# B&R Automation Studio project PLC code - cp (part 12)

#### BlockAlarms.st
```iecst
ACTION BlockAlarms:

	// Report alrms if is enabled. It comes from 4.3.6
	IF NOT Block.Status.xEnabledMovements THEN
		// Emergency stop alarm report to SW with block disabled
		SafetyEmergencyStopAlarms;
		RETURN;
	END_IF

	SafetyAlarms;

	ModulesElementsAlarms;

	VerticalMotorAlarms;

	CleanAlarms;

	//########################## ALARMS SUMMARY ########################################
	AlarmsSummary;

END_ACTION

ACTION SafetyAlarms:

	SafetyEmergencyStopAlarms;

	// Alarm: Curtain Alarm

	//[RGP]CRETALEGO-1297: Front curtain alarm always activated when conditions are TRUE. Not autoreset as previously.
	//Will be reset BY "ResetAlarms.st" when "Reset" button is pressed and conditions are no longer TRUE.
	//These lines have been moved up, before calling "T_SafetyError()", this way we can set the alarm before switching to ZERO state
	IF NOT Block.In.Safety.xCurtainEnable01 OR NOT Block.In.Safety.xCurtainEnable02 THEN
		Block.Al.xAlrFrontCurtain:= TRUE;
	END_IF

	//Alarm: Front and rear general alarm (from preventa)
	IF (NOT Block.In.Safety.xRearSafetyOK) THEN
		Block.Al.xAlrRearSafety:= TRUE;
	END_IF
	IF (NOT Block.In.Safety.xFrontSafetyOK) THEN
		Block.Al.xAlrFrontSafety:= TRUE;
	END_IF

	//Bars Out sensor Cube
	IF NOT Block.In.xBarsIn AND Block.Status.Motor.xBarsHomed THEN
		Block.Al.xAlrBarsOut := TRUE;
	END_IF

	//Any Upper Safety. Variable to better readin and reduce number of lines
	xAnyUpperSafety := Block.Al.xAlrFrontCurtain OR Block.Al.xAlrRearSafety OR Block.Al.xAlrFrontSafety OR Block.Al.xAlrBarsOut;

	// Safety feedback is down? Has it been validate by reset panel?
	//Used a TOF to avoid false signal when entering in AutoMode ALX check in P4 this functionallity
	T_SafetyError.IN:=	(NOT Block.commands.Mode.xZero) AND
						(xAnyUpperSafety OR Block.Al.xAlrEmergencyStop OR NOT Block.In.Safety.xSafetyOK) AND
						(NOT Block.commands.AutoMode.xBypass);

	T_SafetyError.PT:=t#150ms;
	T_SafetyError();

	IF T_SafetyError.Q THEN
		Block.Al.xAlrSafetySystemInBlock:= TRUE;
	END_IF

END_ACTION

ACTION SafetyEmergencyStopAlarms:

	CASE Block.parameters.Hw.SafetySignals OF
		SAFETY_ESTOP_CONNECTED:

			// Alarm: Emergency Stop Button
			IF NOT Block.In.Safety.xFrontEStopOK THEN
				Block.Al.xAlrFrontEmergencyStop := TRUE;
			END_IF

			IF NOT Block.In.Safety.xRearEStopOK THEN
				Block.Al.xAlrRearEmergencyStop:= TRUE;
			END_IF

			Block.Al.xAlrEmergencyStop := Block.Al.xAlrFrontEmergencyStop OR Block.Al.xAlrRearEmergencyStop;

		SAFETY_ESTOP_CALCULATED:

			//If we do not have Safety OK buy the upper safety is OK, it is considered and EStop button is pressed
			IF NOT Block.In.Safety.xSafetyOK AND Block.In.Safety.xFrontSafetyOK AND Block.In.Safety.xRearSafetyOK THEN
				Block.Al.xAlrLogicEmergencyStop:= TRUE;
			END_IF

			Block.Al.xAlrEmergencyStop := Block.Al.xAlrLogicEmergencyStop;

	END_CASE

END_ACTION

ACTION VerticalMotorAlarms:

	// Alarm: Not homed Vertical motor.
	Block.Al.xAlrBarMtrNoRef:= NOT Block.Status.Motor.xBarsHomed;

	// Alarm: Drive protection
	IF NOT Block.In.xDriveProtectionOK THEN
		Block.Al.xAlrDriveProtection:= TRUE;
	END_IF

	// Alarm: Temp Vertical Motor
	IF AxisBK.Status.ActTempMot > (AxisBK.Status.MaxTempMotor - 5.0) THEN
		Block.Al.xBarMotorTemp := TRUE;
	ELSIF AxisBK.Status.ActTempMot < (AxisBK.Status.MaxTempMotor - 7.0) THEN
		Block.Al.xBarMotorTemp := FALSE;
	END_IF

	// Alarm: Temp Vertical Driver
	IF AxisBK.Status.ActTempDrv > (AxisBK.Status.MaxTempDrv - 5.0) THEN
		Block.Al.xBarDriverTemp := TRUE;
	ELSIF AxisBK.Status.ActTempDrv < (AxisBK.Status.MaxTempDrv - 7.0) THEN
		Block.Al.xBarDriverTemp := FALSE;
	END_IF

	//Alarm: Comms error in Vertical motor
	// Pass codes to ennum type 32189
	IF (AxisBK.Status.ErrorID=29265) OR (AxisBK.Status.ErrorID=32189) THEN
		Block.Al.xAlrComBarMtr:= TRUE;
	END_IF

	// Alarm: Any drive Alarm
	TON_DelayAnyVerticalDriveAlarm.IN:= AxisBK.Status.ErrorID<>0 AND
										NOT Block.AlSummary.xAlrSafetySystemGeneral AND
										NOT Block.commands.Mode.xZero AND
										NOT xAnyUpperSafety;
	TON_DelayAnyVerticalDriveAlarm.PT:=t#200ms;
	TON_DelayAnyVerticalDriveAlarm();
	IF TON_DelayAnyVerticalDriveAlarm.Q THEN
		ReasonErrorID := AxisBK.Status.ErrorID;
		Block.Al.xAnyVerticalDriveAlarm:= TRUE;
	END_IF

	// Alarm: Power Error
	//[RGP] Power mains: At least one phase of the power line failed
	IF AxisBK.Status.ErrorID=7215 THEN
		Block.Al.xAlBarMotorPowerOff:= TRUE;
	END_IF

	// Warning: Decrease clean offset.
	TOF_CleanOffsetChng.IN := rOffseCleanMtr <> rOffseCleanMtr_Copy;
	TOF_CleanOffsetChng.PT := t#10s;
	TOF_CleanOffsetChng();
	Block.Al.xAlrDecreaseCleanOffset:= TOF_CleanOffsetChng.Q;

	//Warning: Check Homing Sensor Broken
	IF Block.Al.xAnyVerticalDriveAlarm AND (Block.Status.PositionState = BLOCKP_HOMING_BAR) THEN
		Block.Al.xAlrCheckHomingSensor:=TRUE;
	END_IF

	// Warning: Vertical motor maxium lifting alarm
	IF rMotorCurrentPos >= Block.parameters.Motor.rSafePosition THEN
		Block.Al.xAlrBlockReachedMaxPosition := TRUE;
	END_IF

	// Warning: Reference incoherence or broken reference sensor wire
	T_DelayAlarmRef.IN:=Block.In.xReferenceDI <> AxisBK.Status.DigitalInputs.RefSwitch;
	T_DelayAlarmRef.PT:=T#500ms;
	T_DelayAlarmRef();

	IF T_DelayAlarmRef.Q THEN
		Block.Al.xAlrReferenceIncoherence := TRUE;
	END_IF

	//Critical: Controller Not Ready
	ton_ControllerReady.IN := (NOT AxisBK.Status.ControllerReady OR AxisBK.Status.ErrorID=6029 OR AxisBK.Status.ErrorID=29216) AND NOT Block.commands.Mode.xZero;	//ErrorID 6029 its for motors with breaker and ControllerReady its general
	ton_ControllerReady.PT := t#300ms;																																//ErrorID 29216 to detect just power wires disconected
	ton_ControllerReady();
	IF ton_ControllerReady.Q THEN
		Block.Al.xAlrControllerNotReady := TRUE;
	END_IF

	//Warning Over Torque
	TON_OvertorqueWarning.IN := ABS(AxisBK.Status.ActTorque) > (Block.Status.Motor.rOperationTorque); //AxisBK.Status.RatedTorque;
	TON_OvertorqueWarning.PT := T#10s; //T#2s;
	TON_OvertorqueWarning();

	IF TON_OvertorqueWarning.Q THEN
		Block.Al.xWrnOverTorq := TRUE;
	END_IF

	// Alarm: Over Torque
	tonOvertorqueAlarm.IN := ABS(AxisBK.Status.ActTorque) > (1.6*Block.Status.Motor.rOperationTorque); //(AxisBK.Status.RatedTorque);
	tonOvertorqueAlarm.PT := T#500ms;	//T#5s;
	tonOvertorqueAlarm();
	IF tonOvertorqueAlarm.Q THEN
		Block.Al.xAlrOverTorque := TRUE;
	END_IF

	//Alarms related to collision between bars and tray
	CASE Block.Status.PositionState OF
		BLOCKP_UNDEFINED,
		BLOCKP_IN_CAP,
		BLOCKP_IN_CLEAN,
		BLOCKP_HOMING_ICLA:
			// Do nothing

		BLOCKP_IN_PRINT:
			//Raise warning and alarm if the tray sensor is disconected while in risk position (below dripping position)
			tonDelayTraySensorError.IN := NOT Block.In.xTrayOut;
			tonDelayTraySensorError.PT := T#750ms;
			tonDelayTraySensorError();

			//Raise asking the machine to emptyBelt
			IF tonDelayTraySensorError.Q AND Block.parameters.xMediaBelow THEN
				Block.Status.xAlarmToEmptyBelt := TRUE;
			//Raise and stop alarm once the belt is empty
			ELSIF tonDelayTraySensorError.Q AND NOT Block.parameters.xMediaBelow THEN
				Block.Al.xAlrTraySensor:=TRUE;
				Block.Status.xAlarmToEmptyBelt := FALSE;
			END_IF

		BLOCKP_GOING_TO_CAP,
		BLOCKP_GOING_TO_PRINT,
		BLOCKP_GOING_TO_CLEAN,
		BLOCKP_CLEANING,
		BLOCKP_HOMING_BAR:
			//Risk. Moving!
			xDangerCollision := NOT Block.In.xTrayOut OR NOT Block.In.xIclaSensor;
			IF NOT Block.In.xTrayOut AND 	(((rMotorCurrentPos<Block.parameters.Motor.rDripBarsPosition) AND NOT Block.parameters.xCappingProcess) OR
												(rMotorCurrentPos<Block.parameters.Motor.rCappingPosition)) OR

				NOT Block.In.xIclaSensor AND (((rMotorCurrentPos<Block.parameters.Motor.rSafePositionCleanCarrier) AND NOT Block.parameters.xCappingProcess) OR
												(rMotorCurrentPos<Block.parameters.Motor.rCappingPosition))	THEN

					Block.Al.xNoActionDangerCollision:=TRUE;
			END_IF
	END_CASE

	//Saving state where alarm was raised
	IF EDGEPOS(Block.Al.xNoActionDangerCollision) THEN
		iReasonDanger.0:=NOT Block.In.xTrayOut;
		iReasonDanger.1:=NOT Block.In.xIclaSensor;

		nStateDanger := nState;
		PositionStateDanger:=Block.Status.PositionState;
	END_IF

	//If the sensor is conected again. Remove the memory
	IF Block.In.xTrayOut THEN
		Block.Status.xAlarmToEmptyBelt := FALSE;
	END_IF

END_ACTION

ACTION ModulesElementsAlarms:

	// Alarm: Differential NOK
	IF NOT Block.In.xDifferentialOK THEN
		Block.Al.xAlrDif:= TRUE;
	END_IF

	// Alarm: TempPowerSupply
	IF Block.parameters.Hw.iNumHeaterPSU>0 THEN
		Block.Al.xAlrTempPowerSupply:= FALSE;
		FOR iIndexPsu:=1 TO Block.parameters.Hw.iNumHeaterPSU DO
			IF NOT Block.In.xHeaterDcOkPsu[iIndexPsu] OR NOT Block.In.xHeaterAcOkPsu[iIndexPsu] THEN
				Block.Al.xAlrTempPowerSupply:= TRUE;
			END_IF
		END_FOR

		IF NOT Block.In.xHeaterDcOkBusBar1 OR NOT Block.In.xHeaterDcOkBusBar2 THEN
			Block.Al.xAlrTempPowerSupply:= TRUE;
		END_IF
	END_IF

	// Logging the exact signal that raises the Heaters Power supply alarm
	IF EDGENEG(Block.In.xHeaterDcOkBusBar1) THEN LogErrorxHeaterDcOkBusBar1; END_IF
	IF EDGENEG(Block.In.xHeaterDcOkBusBar2) THEN LogErrorxHeaterDcOkBusBar2; END_IF
	IF EDGENEG(Block.In.xHeaterDcOkPsu[1]) THEN LogErrorxHeaterDcOkPsu1; END_IF
	IF EDGENEG(Block.In.xHeaterDcOkPsu[2]) THEN LogErrorxHeaterDcOkPsu2; END_IF
	IF EDGENEG(Block.In.xHeaterDcOkPsu[3]) THEN LogErrorxHeaterDcOkPsu3; END_IF
	IF EDGENEG(Block.In.xHeaterAcOkPsu[1]) THEN LogErrorxHeaterAcOkPsu1; END_IF
	IF EDGENEG(Block.In.xHeaterAcOkPsu[2]) THEN LogErrorxHeaterAcOkPsu2; END_IF
	IF EDGENEG(Block.In.xHeaterAcOkPsu[3]) THEN LogErrorxHeaterAcOkPsu3; END_IF

	// Alarm: PrintHead PowerSupply
	IF Block.parameters.Hw.iNumPrintheadsPSU>0 THEN
		Block.Al.xAlrPHPowerSupply:= FALSE;
		FOR iIndexPsu:=1 TO Block.parameters.Hw.iNumPrintheadsPSU DO
			IF NOT Block.In.xPrintHeadPSU[iIndexPsu] THEN
				Block.Al.xAlrPHPowerSupply:= TRUE;
			END_IF
		END_FOR
	END_IF

	// Alarm: Module Temp 01
	Block.Al.xModuleTemp01:= NOT Block.In.xModuleTemp01Ok;

	// Alarm: Module Temp 02
	Block.Al.xModuleTemp02:= NOT Block.In.xModuleTemp02Ok;

	// Alarm: Module Temp 03
	Block.Al.xModuleTemp03:= NOT Block.In.xModuleTemp03Ok AND Block.parameters.Inks.xTankHeatEnabled1;

	// Alarm: Module Temp 04
	Block.Al.xModuleTemp04:= NOT Block.In.xModuleTemp04Ok AND Block.parameters.Inks.xTankHeatEnabled2;

	(*SI UNIT ALARMS*)
	//Alarm venturi
	IF NOT Block.In.xAirVenturiOK AND Block.In.xSiUnitModuleOk THEN
		Block.Al.xAlAirVenturi:= TRUE;
	END_IF

	// Alarm: Coms error SI Unit
	IF NOT Block.In.xSiUnitModuleOk  THEN
		Block.Al.xAlrComSiUnit:= TRUE;
		Block.Al.xSiUnitPowerOff:=TRUE;
	END_IF

END_ACTION

ACTION CleanAlarms:

	// Warning: Alarms of no action allowed due to colision warning.
	Block.Al.xAlrNoTrayInServoNoHomed:=(NOT AxisBK.Status.HomeOK) AND Block.commands.Manual.xManTrayIn;

	// Warning: clean interrupt
	Block.Al.xAlCleanInterrupt:= xCleanInterrupt;

	// ICLA		ICLA		ICLA		ICLA		ICLA		ICLA		ICLA		ICLA
	// ICLA		ICLA		ICLA		ICLA		ICLA		ICLA		ICLA		ICLA

	//Alarm: Comms error in cleaning motor
	T_AlrComsCleanMotor.IN:= NOT IclaBK.Status.xModuleOK;
	T_AlrComsCleanMotor.PT:= T#2S;
	T_AlrComsCleanMotor();

	IF T_AlrComsCleanMotor.Q THEN
		Block.Al.xAlrComCleanMtr:= TRUE;
	END_IF

	//Alarm: Not homed cleaning motor.
	Block.Al.xAlrCleanMtrNoRef:= NOT Block.Status.Icla.xHomed;

	// From Icla error table 011Ah 282 4 Inputs of the STO safety function have different levels (>1s). Reset done executing ResetAlarms in Machine program
	// If the connector is removed while moving is error 281, error 282 is STO at different level
	IF (IclaBK.Status.Error.ErrorNumber = 281 OR IclaBK.Status.Error.ErrorNumber = 282) THEN
		Block.Al.xAlrEnabCleanMtrDiffLvL:= TRUE;
	END_IF

	// Alarm: Any clean motor alarm
	T_IclaError.IN :=	(IclaBK.Status.Error.ErrorNumber<>0 OR IclaBK.Status.iDriveStatus = ICLAST_SWITCH_ON_DISABLED OR IclaBK.Status.iDriveStatus = ICLAST_ERROR) AND
						Block.In.Safety.xSafetyOK AND
						NOT Block.AlSummary.xAlrSafetySystemGeneral AND //This variable must not be required so we already check "Block.In.Safety.xSafetyOK"
						NOT Block.commands.Mode.xZero AND
						NOT xAnyUpperSafety; //This variable must not be required so we already check "Block.In.Safety.xSafetyOK"
	T_IclaError.PT := t#250ms;
	T_IclaError();
	IF T_IclaError.Q THEN
		Block.Al.xAlrCleanMotor:= TRUE;
	END_IF

	Block.Al.xCleanMotorControllerNotReady := IclaBK.Status.iDriveStatus = ICLAST_SWITCH_ON_DISABLED AND Block.In.Safety.xSafetyOK AND NOT Block.commands.Mode.xZero;

	// Alarm: Clean Sensor
	T_AlCleanSensor.IN:= Block.Status.Icla.xHomed AND (NOT Block.In.xIclaSensor) AND (rIclaCurrentPos<=0) AND Block.In.xSiUnitModuleOk;
	T_AlCleanSensor.PT:= t#2500ms;
	T_AlCleanSensor();
	IF T_AlCleanSensor.Q THEN
		Block.Al.xAlrCleanSensor:= TRUE;
	END_IF

	// TRAY ALARMS		TRAY ALARMS		TRAY ALARMS		TRAY ALARMS		TRAY ALARMS		TRAY ALARMS		TRAY ALARMS		TRAY ALARMS
	// TRAY ALARMS		TRAY ALARMS		TRAY ALARMS		TRAY ALARMS		TRAY ALARMS		TRAY ALARMS		TRAY ALARMS		TRAY ALARMS

	TNotPrinterZero.IN:=NOT (Block.commands.Mode.xZero);
	TNotPrinterZero.PT:=T#500ms;
	TNotPrinterZero();

	//This is to avoid alarms in Zero mode when manually moving the tray
	IF TNotPrinterZero.Q THEN
		TON_AlrTrayIn(IN := Block.Out.xTrayIn, PT:= Block.parameters.tiTimeWaitTrayInAlarm);
		TON_AlrTrayOut(IN := Block.Out.xTrayOut, PT:= Block.parameters.tiTimeWaitTrayOutAlarm);
	END_IF

	// Alr tray sensor IN
	IF TON_AlrTrayIn.Q AND (NOT Block.In.xTrayIn) THEN
		Block.Al.xAlrTraySensor:=TRUE;
	END_IF
	// Alr tray sensor OUT
	IF TON_AlrTrayOut.Q AND (NOT Block.In.xTrayOut) THEN
		Block.Al.xAlrTraySensor:=TRUE;
	END_IF

	//Alarm clean motor ERROR POSITION// issue 1269
	T_DelayIncoherCleanMtr.IN :=	((nState=233 AND NOT Block.In.xIclaSensor) OR
									(rIclaCurrentPos>LIMITPOSINCOHERCLEANMOTOR AND Block.In.xIclaSensor));
	T_DelayIncoherCleanMtr.PT:= T#500MS;
	T_DelayIncoherCleanMtr();

	IF T_DelayIncoherCleanMtr.Q THEN
		Block.Al.xAlrIncoherPositCleanMtr:= TRUE;
	END_IF
	//Poner aquí la gestion de las alarmas y, si eso, sacar la habilitación fuera, ya que no es su sitio
	//Secuencia - Alarmas de tanque y bomba - Sirena - Hab/Deshab - parada a mitad de proceso - ....

	//If Machine are Water enable water alarms
	IF Block.Status.xIsWaterBlock THEN

		//Water tank empty alarm
		IF NOT Block.In.xWaterLevelSensor THEN
			Block.Al.xAlrEmptyWaterTank:=TRUE;
		END_IF

		//Water Presure and broken presure sensor alarms
		T_AlrNoPressureWhenWaterPumpIsOn.IN:=Block.Out.xCleaningWaterPump AND Block.In.xWaterPresureSensor;
		T_AlrNoPressureWhenWaterPumpIsOn.PT:=T#5S;
		T_AlrNoPressureWhenWaterPumpIsOn();
		IF T_AlrNoPressureWhenWaterPumpIsOn.Q THEN
			Block.Al.xAlrWaterPumpPresure:=TRUE;
		END_IF

		//Broquen wire or pressure switch not work alarm
		IF NOT Block.In.xWaterPresureSensor AND NOT Block.Out.xCleaningWaterPump AND NOT nState=264 THEN
			Block.Al.xAlrWtrPresSensBroken := TRUE;
		END_IF

		//Capping water Alarms:
		//Water flowmeter and WaterTankEmpty
		IF Block.parameters.xCappingProcess  THEN

			//Water tank empty alarm
			IF NOT Block.In.xCappingWaterLevelSensor THEN
				Block.Al.xAlrCappingWaterTankEmpty:=TRUE;
			END_IF

			//Water recirculation alarm
			TON_AlrCappingWaterNotRecirc.IN:=(Block.Out.xCappingWaterPump AND NOT Block.In.xCappingWaterFlowmeter);
			TON_AlrCappingWaterNotRecirc.PT:=T#3S;
			TON_AlrCappingWaterNotRecirc();

			IF TON_AlrCappingWaterNotRecirc.Q THEN
				//Block.Al.xAlrCappingWaterNotRecirc:=TRUE;
			END_IF
		END_IF

	END_IF

	xAlrToAvoidCleanWithWater := Block.Al.xAlrEmptyWaterTank OR Block.Al.xAlrWaterPumpPresure OR Block.Al.xAlrWtrPresSensBroken;

END_ACTION
```

#### BlockManager.st
```iecst
PROGRAM _INIT
	FOR iIndexHistory:=0  TO iHistoryLines DO
		StateGenHistory[iIndexHistory]:=BLOCK_STOPPED;
		StatePosHistory[iIndexHistory]:=BLOCKP_UNDEFINED;
	END_FOR
END_PROGRAM

(*
PROGRAM _INIT

	//Define a transmision data to do the first calculations and be receptive to next calculations
	MotorDriveUnit.TransmissionData:=Block.parameters.Motor.DriveUnit;

	//Acceleration and deceleration
	MotorDriveUnit.AccelerationDesired := 10;
	MotorDriveUnit.Calculation := CALC_ACC_PULSES;
	MotorDriveUnit();

	MotorDriveUnit.DecelerationDesired := 10;
	MotorDriveUnit.Calculation := CALC_DEC_PULSES;
	MotorDriveUnit();

END_PROGRAM
*)

PROGRAM _CYCLIC

	// Block Reference
	Block ACCESS ADR(gBlock[gIndexBlock]);
	AxisBK ACCESS ADR (gAxis[Block.parameters.iMotorAxisIndex]);
	IclaBK ACCESS ADR (gIcla[Block.parameters.iIclaAxisIndex]);

	//If the Block doesn't exist, remove alarms and exit. Extra condition to avoid a divided by 0 error at start
	IF NOT Block.parameters.Hw.xExistBlock OR Block.parameters.Inks.iMaxBlockPrintBars = 0 THEN
		ResetAlarms;
		ResetBlockCommands;
		gIndexBlock := gIndexBlock + 1;
		RETURN;
	END_IF

	Inputs;

	//Limit the value of parameters configured
	BlockParameters;

	IF Block.parSw.xEnableToMovements THEN
		Block.Status.xEnabledMovements:= TRUE;
	ELSIF NOT Block.parSw.xEnableToMovements AND (xInCap OR NOT Block.Status.Motor.xBarsHomed) THEN
		Block.Status.xEnabledMovements:= FALSE;
	END_IF

	IF Block.commands.xReset THEN
		ResetAlarms;
	END_IF

	BlockAlarms;
	AlarmSound;

	IF (NOT Block.Status.xEnabledMovements) THEN
		gIndexBlock := gIndexBlock + 1;
		RETURN;
	END_IF

	GetInkSystemsData;

	ControlState;

	BlockStatesCtrl;

	AssignDataToInksSystem;

	InputParamsMotors;

	//Managment of the valves unit of the block. Reset if needed
	ValvesUnit;

	//Copy of variables to check changes
	rOffseCleanMtr_Copy:=rOffseCleanMtr;

	ResetEdgeCommands;

	//Increased exec times number to be checked outside
	Block.Status.execTimes := Block.Status.execTimes + 1;

	// Index added
	gIndexBlock := gIndexBlock + 1;

END_PROGRAM
```

#### BlockStateGen.st
```iecst
ACTION BlockStateGen:

	// PRINT POSITION ORDER
	xOrderToPrint:=	(Block.commands.xToPrint AND Block.parSw.xEnableToPrint) OR
					(Block.commands.xToPrintLab AND Block.commands.AutoMode.xLaboratory);

	// CAP POSITION ORDER
	//When in capping position, bars are touching the tray and was required to be able to move out bars in auto mode when front doors is opened
	IF Block.Status.Position.xInCap AND Block.parameters.xCappingProcess THEN
		xFrontDoorStatusChanged := (Block.In.xFrontDoorClosed <> xFrontDoorStatus) OR
									(NOT Block.In.xFrontDoorClosed AND EDGEPOS(Block.commands.Mode.xAuto));
	END_IF

	xCapOrder:= Block.commands.xToCap OR
				(Block.commands.xToCapLab AND Block.commands.AutoMode.xLaboratory) OR
				EDGENEG(Block.parSw.xEnableToPrint) OR
				xFrontDoorStatusChanged;

	xFrontDoorStatus := Block.In.xFrontDoorClosed;

	// CLEANING CYCLE FROM SW COMMAND
	Block.Status.xIsWaterBlock := Block.parameters.Hw.xIsWater AND Block.commands.xEnableCleaningWithWater;
	IF Block.Status.xIsWaterBlock AND xAlrToAvoidCleanWithWater THEN
		Block.Status.xEnabledToClean := FALSE;
	ELSE
		Block.Status.xEnabledToClean := TRUE;
	END_IF

	rsCleaning.SET:= Block.Status.xEnabledToClean AND
					(Block.commands.xStartToCleanOrder AND Block.Status.PositionState <> BLOCKP_CLEANING);
	rsCleaning.RESET1:= NOT Block.Status.xEnabledToClean OR
						EDGEPOS(Block.Status.xCleaningDone) OR
						NOT (Block.commands.Mode.xAuto);
	rsCleaning();
	xStartToCleanOrder:=rsCleaning.Q1;

	//To reset manual commands when not in manual mode
	IF Block.Status.BlockState <> BLOCK_MANUAL THEN
		Block.commands.Manual := ResetManCommands;
	END_IF

	CASE Block.Status.BlockState OF

		BLOCK_STOPPED:
			AxisBK.Command.QuickStop:=FALSE;

		BLOCK_STOPPING:
			StopMovements;
			//Added to modify block position so for example when homing icla or bar and
			//going TO zero, block position remained in homing even motors were stopped and Block status were "BLOCK_STOPPING"
			IF (Block.Status.PositionState=BLOCKP_HOMING_ICLA OR Block.Status.PositionState=BLOCKP_HOMING_BAR) THEN
				Block.Status.PositionState := BLOCKP_UNDEFINED;
			END_IF

			IF AllDevicedStopped(ADR(Block), ADR(AxisBK), ADR(IclaBK)) THEN
				Block.Status.BlockState := BLOCK_STOPPED;
			END_IF

		BLOCK_MANUAL:
			ManualMovements;

			IF Block.commands.xIclaHomeOrder AND NOT Block.Status.Motor.xBarsHoming THEN
				IF Block.parameters.xPrinterKeyMaintenanceActivated THEN
					Block.commands.xIclaHomeOrder:=FALSE;
				ELSE
					Block.Status.PositionState := BLOCKP_HOMING_ICLA;
				END_IF

			// To do home in block is mandatory to have Icla at sensor and try out
			ELSIF Block.commands.xBarHomeOrder THEN

				IF Block.In.xTrayIn OR NOT Block.In.xIclaSensor OR Block.parameters.xPrinterKeyMaintenanceActivated THEN
					Block.commands.xBarHomeOrder:=FALSE;
				ELSIF Block.In.xTrayOut AND Block.In.xIclaSensor AND NOT Block.Al.xAlrReferenceIncoherence THEN
					Block.Status.PositionState := BLOCKP_HOMING_BAR;
				ELSE
					Block.commands.xBarHomeOrder:=FALSE;
				END_IF

			ELSIF Block.commands.xToCleanPosition AND Block.Status.PositionState = BLOCKP_IN_CAP THEN
				Block.Status.PositionState := BLOCKP_GOING_TO_CLEAN;
				//Signal reseted outside the case to avoid a memory if the movement cannot be done

			ELSIF Block.commands.Manual.xToPrintPosition AND NOT Block.parameters.xMediaBelow AND Block.Status.PositionState = BLOCKP_IN_CAP THEN
				Block.Status.PositionState := BLOCKP_GOING_TO_PRINT;
				//Signal reseted outside the case to avoid a memory if the movement cannot be done

			END_IF

		BLOCK_AUTO:
			IF xStartToCleanOrder THEN

				//Enable cleaning in bar to end ReverseFlow
				IF Block.Status.PositionState <> BLOCKP_CLEANING THEN
					IF 	Block.Status.PositionState = BLOCKP_GOING_TO_PRINT OR Block.Status.PositionState = BLOCKP_IN_PRINT THEN
						BlockPositionPreviousCleaning := BLOCKP_GOING_TO_PRINT;
					ELSE
						BlockPositionPreviousCleaning := BLOCKP_GOING_TO_CAP;
					END_IF
					Block.Status.PositionState := BLOCKP_CLEANING;
				END_IF

				//If receiving a Going to Cap order while cleaning, store the information
				IF xCapOrder THEN
					BlockPositionPreviousCleaning := BLOCKP_GOING_TO_CAP;
				END_IF

			ELSIF (xCapOrder AND Block.Status.Motor.xBarsHomed AND (Block.In.xIclaSensor OR IclaBK.Status.iDriveStatus=ICLAST_ENABLE_OPERATION)) THEN
				//I move to STOP
				Block.Status.PositionState := BLOCKP_GOING_TO_CAP;

			ELSIF xOrderToPrint AND NOT xInPrint AND NOT Block.AlSummary.xAlarmCritical AND NOT Block.AlSummary.xAlarmStop THEN
				//Going TO PRINT
				Block.Status.PositionState := BLOCKP_GOING_TO_PRINT;

			END_IF

			IF 	EDGEPOS(Block.Status.xCleaningDone) THEN
				//Once he cleaning has finished, go to the previous position
				Block.Status.PositionState := BlockPositionPreviousCleaning;
			END_IF

	END_CASE

	//Copying block's outputs to status
	Block.Status.ManualCommands := Block.Out;

	//Saving state history
	IF Block.Status.BlockState<>StateGenHistory[0] THEN
		ShiftArrayForward(ADR(StateGenHistory), SIZEOF(StateGenHistory), SIZEOF(StateGenHistory[0]), 1, iHistoryLines);
		StateGenHistory[0]:=Block.Status.BlockState;
	END_IF

END_ACTION
```

#### EventLog.st
```iecst
ACTION LogCriticalAlarm:

//	iReasonCritical.0 := (Block.Al.xAlrSafetySystemInBlock AND Block.Status.xEnabledMovements);
//	iReasonCritical.1 := Block.Al.xAlrDif;
//	iReasonCritical.2 := Block.Al.xAlrDriveProtection;

	stEventLogCritical.Source := ELOG_TYPE_BLOCK;
	stEventLogCritical.Severity:= ELOG_SEVERITY_ERROR;
	stEventLogCritical.Facility:= gIndexBlock;
	stEventLogCritical.ErrorCode:=0;

	stEventLogCritical.Text := 'Block.LogCriticalAlarm';

	IF 		iReasonCritical.0 THEN stEventLogCritical.Text := 'Block. xAlrSafetySystemInBlock';
	ELSIF 	iReasonCritical.1 THEN stEventLogCritical.Text := 'Block. xAlrDif';
	ELSIF 	iReasonCritical.2 THEN stEventLogCritical.Text := 'Block. xAlrDriveProtection';
	END_IF

	gEventLogLoader(EventData := ADR(stEventLogCritical));

END_ACTION

ACTION LogStopAlarm:

	stEventLogStop.Source := ELOG_TYPE_BLOCK;
	stEventLogStop.Severity:= ELOG_SEVERITY_ERROR;
	stEventLogStop.Facility:= gIndexBlock;
	stEventLogStop.ErrorCode:=0;

	stEventLogStop.Text := 'Block.LogStopAlarm';

	IF 		iReasonStop.0 THEN stEventLogStop.Text := 'Block. xAlrCleanMtrNoRef';
	ELSIF 	iReasonStop.1 THEN stEventLogStop.Text := 'Block. xAlAirVenturi';
	ELSIF 	iReasonStop.2 THEN stEventLogStop.Text := 'Block. xAnyDriveAlarm';
	ELSIF 	iReasonStop.3 THEN stEventLogStop.Text := 'Block. xAlrBarMtrNoRef';
	ELSIF 	iReasonStop.4 THEN stEventLogStop.Text := 'Block. xSiUnitPowerOff';
	ELSIF 	iReasonStop.5 THEN stEventLogStop.Text := 'Block. xAlrComSiUnit';
	ELSIF 	iReasonStop.6 THEN stEventLogStop.Text := 'Block. xAlrComBarMtr';
	ELSIF 	iReasonStop.7 THEN stEventLogStop.Text := 'Block. xAlrCleanMotor';
	ELSIF 	iReasonStop.8 THEN stEventLogStop.Text := 'Block. xAlrComCleanMtr';
	ELSIF 	iReasonStop.9 THEN stEventLogStop.Text := 'Block. xAlrEnabCleanMtrDiffLvL';
	ELSIF 	iReasonStop.10 THEN stEventLogStop.Text := 'Block. xAlrIncoherPositCleanMtr';
	ELSIF 	iReasonStop.11 THEN stEventLogStop.Text := 'Block. xAlCleanInterrupt';
	ELSIF 	iReasonStop.12 THEN stEventLogStop.Text := 'Block. xAlrTrayCleanSensor';
	ELSIF 	iReasonStop.13 THEN stEventLogStop.Text := 'Block. xNoActionDangerCollision';
	ELSIF 	iReasonStop.14 THEN stEventLogStop.Text := 'Block. xAlrControllerNotReady';
	ELSIF 	iReasonStop.15 THEN stEventLogStop.Text := 'Block. xAlrOverTorque';
	END_IF

	//Adding nState data to log
	strAuxEventDesc := '. nSt= ';
	brsstrcat(ADR(stEventLogStop.Text), ADR(strAuxEventDesc));
	brsitoa(nState, ADR(strAuxEventDesc));
	brsstrcat(ADR(stEventLogStop.Text), ADR(strAuxEventDesc));
	strAuxEventDesc := '. nDg= ';
	brsstrcat(ADR(stEventLogStop.Text), ADR(strAuxEventDesc));
	brsitoa(nStateDanger, ADR(strAuxEventDesc));
	brsstrcat(ADR(stEventLogStop.Text), ADR(strAuxEventDesc));

	gEventLogLoader(EventData := ADR(stEventLogStop));

END_ACTION

ACTION LogToCapOrder:

	stEventLogToCap.Source := ELOG_TYPE_BLOCK;
	stEventLogToCap.Severity:= ELOG_SEVERITY_INFO;
	stEventLogToCap.Facility:= gIndexBlock;
	stEventLogToCap.ErrorCode:=0;

	stEventLogToCap.Text := 'Order to Cap BK: ';
	brsitoa(gIndexBlock, ADR(strAuxEventDesc));
	brsstrcat(ADR(stEventLogToCap.Text), ADR(strAuxEventDesc));

	gEventLogLoader(EventData := ADR(stEventLogToCap));

END_ACTION

ACTION LogToPrintOrder:

	stEventLogToPrint.Source := ELOG_TYPE_BLOCK;
	stEventLogToPrint.Severity:= ELOG_SEVERITY_INFO;
	stEventLogToPrint.Facility:= gIndexBlock;
	stEventLogToPrint.ErrorCode:=0;

	stEventLogToPrint.Text := 'Order to Print BK: ';
	brsitoa(gIndexBlock, ADR(strAuxEventDesc));
	brsstrcat(ADR(stEventLogToPrint.Text), ADR(strAuxEventDesc));

	gEventLogLoader(EventData := ADR(stEventLogToPrint));

END_ACTION

ACTION LogToCleanOrder:

	stEventLogToClean.Source := ELOG_TYPE_BLOCK;
	stEventLogToClean.Severity:= ELOG_SEVERITY_INFO;
	stEventLogToClean.Facility:= gIndexBlock;
	stEventLogToClean.ErrorCode:=0;

	stEventLogToClean.Text := 'Order to Clean BK: ';
	brsitoa(gIndexBlock, ADR(strAuxEventDesc));
	brsstrcat(ADR(stEventLogToClean.Text), ADR(strAuxEventDesc));

	gEventLogLoader(EventData := ADR(stEventLogToClean));

END_ACTION

ACTION LogVertMovementOrder:

	VerMotorEventLog.Source := ELOG_TYPE_BLOCK;
	VerMotorEventLog.Severity:= ELOG_SEVERITY_INFO;
	VerMotorEventLog.Facility:= gIndexBlock;
	VerMotorEventLog.ErrorCode:=0;

	VerMotorEventLog.Text := 'BK:';
	brsitoa(gIndexBlock, ADR(strAuxEventDesc));
	brsstrcat(ADR(VerMotorEventLog.Text), ADR(strAuxEventDesc));

	brsstrcat(ADR(VerMotorEventLog.Text), ADR(' from '));
	brsftoa(MotorDriveUnit.PositionDevice, ADR(strAuxEventDesc));
	brsstrcat(ADR(VerMotorEventLog.Text), ADR(strAuxEventDesc));

	brsstrcat(ADR(VerMotorEventLog.Text), ADR('mm to '));
	brsftoa(MotorDriveUnit.PositionDesired, ADR(strAuxEventDesc));
	brsstrcat(ADR(VerMotorEventLog.Text), ADR(strAuxEventDesc));

	brsstrcat(ADR(VerMotorEventLog.Text), ADR('mm at '));
	brsftoa(MotorDriveUnit.SpeedDesired, ADR(strAuxEventDesc));
	brsstrcat(ADR(VerMotorEventLog.Text), ADR(strAuxEventDesc));

	brsstrcat(ADR(VerMotorEventLog.Text), ADR('mm/s. St: '));
	brsitoa(nState, ADR(strAuxEventDesc));
	brsstrcat(ADR(VerMotorEventLog.Text), ADR(strAuxEventDesc));

	gEventLogLoader(EventData := ADR(VerMotorEventLog));

END_ACTION

ACTION LogVertInPosition:

	VerMotorEventLog.Source := ELOG_TYPE_BLOCK;
	VerMotorEventLog.Severity:= ELOG_SEVERITY_INFO;
	VerMotorEventLog.Facility:= gIndexBlock;
	VerMotorEventLog.ErrorCode:=0;

	VerMotorEventLog.Text := 'In Position BK ';
	brsitoa(gIndexBlock, ADR(strAuxEventDesc));
	brsstrcat(ADR(VerMotorEventLog.Text), ADR(strAuxEventDesc));
	brsstrcat(ADR(VerMotorEventLog.Text), ADR(': '));
	brsftoa(MotorDriveUnit.PositionDevice, ADR(strAuxEventDesc));
	brsstrcat(ADR(VerMotorEventLog.Text), ADR(strAuxEventDesc));
	brsstrcat(ADR(VerMotorEventLog.Text), ADR('mm. St: '));
	brsitoa(nState, ADR(strAuxEventDesc));
	brsstrcat(ADR(VerMotorEventLog.Text), ADR(strAuxEventDesc));

	gEventLogLoader(EventData := ADR(VerMotorEventLog));

END_ACTION

ACTION LogIclaMovementOrder:

	stIclaOrderEventLog.Source := ELOG_TYPE_BLOCK;
	stIclaOrderEventLog.Severity:= ELOG_SEVERITY_INFO;
	stIclaOrderEventLog.Facility:= gIndexBlock;
	stIclaOrderEventLog.ErrorCode:=0;

	stIclaOrderEventLog.Text := 'Icla Order BK: ';
	brsitoa(gIndexBlock, ADR(strAuxEventDesc));
	brsstrcat(ADR(stIclaOrderEventLog.Text), ADR(strAuxEventDesc));
	brsstrcat(ADR(stIclaOrderEventLog.Text), ADR(': '));
	brsftoa(IclaDriveUnit.PositionDesired, ADR(strAuxEventDesc));
	brsstrcat(ADR(stIclaOrderEventLog.Text), ADR(strAuxEventDesc));
	brsstrcat(ADR(stIclaOrderEventLog.Text), ADR('mm. St: '));
	brsitoa(nState, ADR(strAuxEventDesc));
	brsstrcat(ADR(stIclaOrderEventLog.Text), ADR(strAuxEventDesc));

	gEventLogLoader(EventData := ADR(stIclaOrderEventLog));

END_ACTION

ACTION LogIclaInPosition:

	stIclaEventLog.Source := ELOG_TYPE_BLOCK;
	stIclaEventLog.Severity:= ELOG_SEVERITY_INFO;
	stIclaEventLog.Facility:= gIndexBlock;
	stIclaEventLog.ErrorCode:=0;

	stIclaEventLog.Text := 'Icla In Position BK: ';
	brsitoa(gIndexBlock, ADR(strAuxEventDesc));
	brsstrcat(ADR(stIclaEventLog.Text), ADR(strAuxEventDesc));
	brsstrcat(ADR(stIclaEventLog.Text), ADR(': '));
	brsftoa(IclaDriveUnit.PositionDevice, ADR(strAuxEventDesc));
	brsstrcat(ADR(stIclaEventLog.Text), ADR(strAuxEventDesc));
	brsstrcat(ADR(stIclaEventLog.Text), ADR('mm. St: '));
	brsitoa(nState, ADR(strAuxEventDesc));
	brsstrcat(ADR(stIclaEventLog.Text), ADR(strAuxEventDesc));

	gEventLogLoader(EventData := ADR(stIclaEventLog));

END_ACTION

ACTION LogHomingOrderBar:

	VerMotorEventLog.Source := ELOG_TYPE_BLOCK;
	VerMotorEventLog.Severity:= ELOG_SEVERITY_INFO;
	VerMotorEventLog.Facility:= gIndexBlock;
	VerMotorEventLog.ErrorCode:=0;

	VerMotorEventLog.Text := 'Homing order Vert BK: ';
	brsitoa(gIndexBlock, ADR(strAuxEventDesc));
	brsstrcat(ADR(VerMotorEventLog.Text), ADR(strAuxEventDesc));

	gEventLogLoader(EventData := ADR(VerMotorEventLog));

END_ACTION

ACTION LogHomedBar:

	VerMotorEventLog.Source := ELOG_TYPE_BLOCK;
	VerMotorEventLog.Severity:= ELOG_SEVERITY_INFO;
	VerMotorEventLog.Facility:= gIndexBlock;
	VerMotorEventLog.ErrorCode:=0;

	VerMotorEventLog.Text := 'Vert Motor Homed BK: ';
	brsitoa(gIndexBlock, ADR(strAuxEventDesc));
	brsstrcat(ADR(VerMotorEventLog.Text), ADR(strAuxEventDesc));

	gEventLogLoader(EventData := ADR(VerMotorEventLog));

END_ACTION

ACTION LogHomingOrderIcla:

	stIclaEventLog.Source := ELOG_TYPE_BLOCK;
	stIclaEventLog.Severity:= ELOG_SEVERITY_INFO;
	stIclaEventLog.Facility:= gIndexBlock;
	stIclaEventLog.ErrorCode:=0;

	stIclaEventLog.Text := 'Homing order Icla BK: ';
	brsitoa(gIndexBlock, ADR(strAuxEventDesc));
	brsstrcat(ADR(stIclaEventLog.Text), ADR(strAuxEventDesc));

	gEventLogLoader(EventData := ADR(stIclaEventLog));

END_ACTION

ACTION LogHomedIcla:

	stIclaEventLog.Source := ELOG_TYPE_BLOCK;
	stIclaEventLog.Severity:= ELOG_SEVERITY_INFO;
	stIclaEventLog.Facility:= gIndexBlock;
	stIclaEventLog.ErrorCode:=0;

	stIclaEventLog.Text := 'Icla Homed BK: ';
	brsitoa(gIndexBlock, ADR(strAuxEventDesc));
	brsstrcat(ADR(stIclaEventLog.Text), ADR(strAuxEventDesc));

	gEventLogLoader(EventData := ADR(stIclaEventLog));

END_ACTION

ACTION LogMotorOrderIncoherencyHaltAndMoveAbsolute:

	stEventLogIncoherence.Source := ELOG_TYPE_BLOCK;
	stEventLogIncoherence.Severity:= ELOG_SEVERITY_INFO;
	stEventLogIncoherence.Facility:= gIndexBlock;
	stEventLogIncoherence.ErrorCode:=0;

	stEventLogIncoherence.Text := 'Incoherency orders. Halt and MoveAbsolute BK: ';
	brsitoa(gIndexBlock, ADR(strAuxEventDesc));
	brsstrcat(ADR(stEventLogIncoherence.Text), ADR(strAuxEventDesc));

	gEventLogLoader(EventData := ADR(stEventLogIncoherence));

END_ACTION

ACTION LogErrorxHeaterDcOkBusBar1:

	stEventLogxHeaterDcOkBusBar1.Source := ELOG_TYPE_BLOCK;
	stEventLogxHeaterDcOkBusBar1.Severity:= ELOG_SEVERITY_INFO;
	stEventLogxHeaterDcOkBusBar1.Facility:= gIndexBlock;
	stEventLogxHeaterDcOkBusBar1.ErrorCode:=0;

	stEventLogxHeaterDcOkBusBar1.Text := 'Error in xHeaterDcOkBusBar1 BK: ';
	brsitoa(gIndexBlock, ADR(strAuxEventDesc));
	brsstrcat(ADR(stIclaEventLog.Text), ADR(strAuxEventDesc));

	gEventLogLoader(EventData := ADR(stIclaEventLog));

END_ACTION

ACTION LogErrorxHeaterDcOkBusBar2:

	stEventLogxHeaterDcOkBusBar2.Source := ELOG_TYPE_BLOCK;
	stEventLogxHeaterDcOkBusBar2.Severity:= ELOG_SEVERITY_INFO;
	stEventLogxHeaterDcOkBusBar2.Facility:= gIndexBlock;
	stEventLogxHeaterDcOkBusBar2.ErrorCode:=0;

	stEventLogxHeaterDcOkBusBar2.Text := 'Error in xHeaterDcOkBusBar2 BK: ';
	brsitoa(gIndexBlock, ADR(strAuxEventDesc));
	brsstrcat(ADR(stIclaEventLog.Text), ADR(strAuxEventDesc));

	gEventLogLoader(EventData := ADR(stIclaEventLog));

END_ACTION

ACTION LogErrorxHeaterDcOkPsu1:

	stEventLogxHeaterDcOkPsu1.Source := ELOG_TYPE_BLOCK;
	stEventLogxHeaterDcOkPsu1.Severity:= ELOG_SEVERITY_INFO;
	stEventLogxHeaterDcOkPsu1.Facility:= gIndexBlock;
	stEventLogxHeaterDcOkPsu1.ErrorCode:=0;

	stEventLogxHeaterDcOkPsu1.Text := 'Error in xHeaterDcOkPsu1 BK: ';
	brsitoa(gIndexBlock, ADR(strAuxEventDesc));
	brsstrcat(ADR(stIclaEventLog.Text), ADR(strAuxEventDesc));

	gEventLogLoader(EventData := ADR(stIclaEventLog));

END_ACTION

ACTION LogErrorxHeaterDcOkPsu2:

	stEventLogxHeaterDcOkPsu2.Source := ELOG_TYPE_BLOCK;
	stEventLogxHeaterDcOkPsu2.Severity:= ELOG_SEVERITY_INFO;
	stEventLogxHeaterDcOkPsu2.Facility:= gIndexBlock;
	stEventLogxHeaterDcOkPsu2.ErrorCode:=0;

	stEventLogxHeaterDcOkPsu2.Text := 'Error in xHeaterDcOkPsu2 BK: ';
	brsitoa(gIndexBlock, ADR(strAuxEventDesc));
	brsstrcat(ADR(stIclaEventLog.Text), ADR(strAuxEventDesc));

	gEventLogLoader(EventData := ADR(stIclaEventLog));

END_ACTION

ACTION LogErrorxHeaterDcOkPsu3:

	stEventLogxHeaterDcOkPsu3.Source := ELOG_TYPE_BLOCK;
	stEventLogxHeaterDcOkPsu3.Severity:= ELOG_SEVERITY_INFO;
	stEventLogxHeaterDcOkPsu3.Facility:= gIndexBlock;
	stEventLogxHeaterDcOkPsu3.ErrorCode:=0;

	stEventLogxHeaterDcOkPsu3.Text := 'Error in xHeaterDcOkPsu3 BK: ';
	brsitoa(gIndexBlock, ADR(strAuxEventDesc));
	brsstrcat(ADR(stIclaEventLog.Text), ADR(strAuxEventDesc));

	gEventLogLoader(EventData := ADR(stIclaEventLog));

END_ACTION

ACTION LogErrorxHeaterAcOkPsu1:

	stEventLogxHeaterAcOkPsu1.Source := ELOG_TYPE_BLOCK;
	stEventLogxHeaterAcOkPsu1.Severity:= ELOG_SEVERITY_INFO;
	stEventLogxHeaterAcOkPsu1.Facility:= gIndexBlock;
	stEventLogxHeaterAcOkPsu1.ErrorCode:=0;

	stEventLogxHeaterAcOkPsu1.Text := 'Error in xHeaterAcOkPsu1 BK: ';
	brsitoa(gIndexBlock, ADR(strAuxEventDesc));
	brsstrcat(ADR(stIclaEventLog.Text), ADR(strAuxEventDesc));

	gEventLogLoader(EventData := ADR(stIclaEventLog));

END_ACTION

ACTION LogErrorxHeaterAcOkPsu2:

	stEventLogxHeaterAcOkPsu2.Source := ELOG_TYPE_BLOCK;
	stEventLogxHeaterAcOkPsu2.Severity:= ELOG_SEVERITY_INFO;
	stEventLogxHeaterAcOkPsu2.Facility:= gIndexBlock;
	stEventLogxHeaterAcOkPsu2.ErrorCode:=0;

	stEventLogxHeaterAcOkPsu2.Text := 'Error in xHeaterAcOkPsu2 BK: ';
	brsitoa(gIndexBlock, ADR(strAuxEventDesc));
	brsstrcat(ADR(stIclaEventLog.Text), ADR(strAuxEventDesc));

	gEventLogLoader(EventData := ADR(stIclaEventLog));

END_ACTION

ACTION LogErrorxHeaterAcOkPsu3:

	stEventLogxHeaterAcOkPsu3.Source := ELOG_TYPE_BLOCK;
	stEventLogxHeaterAcOkPsu3.Severity:= ELOG_SEVERITY_INFO;
	stEventLogxHeaterAcOkPsu3.Facility:= gIndexBlock;
	stEventLogxHeaterAcOkPsu3.ErrorCode:=0;

	stEventLogxHeaterAcOkPsu3.Text := 'Error in xHeaterAcOkPsu3 BK: ';
	brsitoa(gIndexBlock, ADR(strAuxEventDesc));
	brsstrcat(ADR(stIclaEventLog.Text), ADR(strAuxEventDesc));

	gEventLogLoader(EventData := ADR(stIclaEventLog));

END_ACTION
```

#### InksGetSet.st
```iecst
ACTION GetInkSystemsData:

	// Vars initialization
	//
	tiDripTimeMax:=0;
	Block.Status.iBarsReadyToPrint:= 0;
	rPowerTempTotalBlock:=0;

	//Running for ALL the bars of the machine. Just will enter for the ones in the block
	FOR iIndexInks:=1 TO Block.parameters.Inks.iMaxMachinePrintBars BY 1 DO

		//To analyze if the PrintBar is from the current block
		IF InkBarInBlock(iIndexInks, ADR(gInks), ADR(Block), gIndexBlock) THEN

			IF gInks[iIndexInks].status.iInkState <> INKS_STOPPED THEN

				// Drip Time Max Calculate for TON_DRIPPING is configured for dripping process
				tiDripTimeMax:=MAX(tiDripTimeMax, gInks[iIndexInks].parSw.tiDripTime);

				// Important: It gives info to block
				IF gInks[iIndexInks].status.xEnabledBarToPrint THEN
					Block.Status.iBarsReadyToPrint:= Block.Status.iBarsReadyToPrint + 1;
				END_IF

			END_IF

			//Calculate power factor reduction
			rPowerTempTotalBlock:= rPowerTempTotalBlock + (gInks[iIndexInks].status.Temp.rDutyCycleTemp/100) * UINT_TO_REAL(gInks[iIndexInks].parameters.parBar.iPowerTempWatt);

		END_IF

	END_FOR;

END_ACTION

ACTION AssignDataToInksSystem:

	// Pending to have 3000 in constants per Block, It is max PSU Power installed in the block
	IF rPowerTempTotalBlock = 0 THEN
		rBlockReductionTempPower := 1.0;
	ELSE
		rBlockReductionTempPower:= UINT_TO_REAL(Block.parameters.Inks.iMaxPSUwattsForBars) / rPowerTempTotalBlock ;
		rBlockReductionTempPower:= MIN(rBlockReductionTempPower, 1.0);
	END_IF

	//Assignation of ink variables
	FOR iIndexInks:=1 TO Block.parameters.Inks.iMaxMachinePrintBars BY 1 DO

		//To analyze if the PrintBar is from the current block
		IF InkBarInBlock(iIndexInks, ADR(gInks), ADR(Block), gIndexBlock) THEN

			gInks[iIndexInks].commands.xOrderCleaning:= Block.commands.xInksOrderCleaning;
			gInks[iIndexInks].commands.xOrderDrip:= Block.commands.xDripControl AND (gInks[iIndexInks].parSw.tiDripTime>0);
			gInks[iIndexInks].commands.xCloseReliefValve := xCloseReliefValve;

			gInks[iIndexInks].parameters.tiDripTimeMax:= tiDripTimeMax;
			gInks[iIndexInks].parameters.Temp.rReductionTempPower:=rBlockReductionTempPower;
			//It allows to work in automatic reverse when block is capped and is configured the command xOnReverseCapped/Idle in the GUI
			gInks[iIndexInks].parameters.xBlockInCap := xInCap;
			//Send to ink sistem when the block is in print position to check the correct ink state to print
			gInks[iIndexInks].parameters.xBlockInPrint := xInPrint;

			//Assigning MaxPrintBarsPerBlock to determine when the printbar can use the PSU to heat the Ink
			gInks[iIndexInks].parameters.Temp.iBarsWithSameBlock:= Block.parameters.Inks.iMaxBlockPrintBars;

		END_IF

	END_FOR;

END_ACTION
```

#### InputParamsMotors.st
```iecst
ACTION InputParamsMotors:

	//ICLA   ICLA   ICLA   ICLA   ICLA   ICLA   ICLA   ICLA   ICLA   ICLA   ICLA   ICLA
	//ICLA   ICLA   ICLA   ICLA   ICLA   ICLA   ICLA   ICLA   ICLA   ICLA   ICLA   ICLA
	//ICLA   ICLA   ICLA   ICLA   ICLA   ICLA   ICLA   ICLA   ICLA   ICLA   ICLA   ICLA

	// PowerOn Command
	IclaBK.Command.Enable:= IclaBK.Status.iDriveStatus <> ICLAST_ERROR AND NOT Block.Al.xAlrSafetySystemInBlock;

	//Just to avoid resetting the Icla when has to move in Automatic mode
	xEnableResetIcla:= Block.Status.PositionState <> BLOCKP_CLEANING;

	// It avoids enables in Icla when Icla is in error state
	IclaBK.Command.Reset:=  NOT Block.Al.xAlrSafetySystemInBlock AND
                            Block.commands.xReset AND
							NOT xIclaMoving AND
							xEnableResetIcla;

	// Block sets Icla Speed in Jog movement
	IclaBK.Parameter.Jog.VeloFast:= 500;
	IclaBK.Parameter.Jog.VeloSlow:= 500;

	// Block sets Icla Speed and positino in Abs movement
	IclaDriveUnit.TransmissionData:=Block.parameters.Icla.DriveUnit;
	IclaDriveUnit.PositionDesired:=rIclaAbsPosDesired;
	IclaDriveUnit.Calculation:=CALC_POS_PULSES;
	IclaDriveUnit();
	IclaBK.Parameter.MoveAbsolute.Position:= REAL_TO_DINT(IclaDriveUnit.pulsesPositionDesired);

	//Just send the information when change
	IF EDGEPOS(xIclaAbsMovOrder) OR EDGENEG(xIclaAbsMovOrder) THEN
		IclaBK.Command.MoveAbsolute:= xIclaAbsMovOrder;
	END_IF
	IF EDGEPOS(xIclaAbsMovOrder) THEN
		LogIclaMovementOrder;
	END_IF

	IclaDriveUnit.pulsesDevice:=DINT_TO_REAL(IclaBK.Status.iActualPosition);
	IclaDriveUnit.Calculation:=CALC_POS_MM;
	IclaDriveUnit();
	Block.Status.Icla.rCurrentPosition:=IclaDriveUnit.PositionDevice;
	rIclaCurrentPos:=IclaDriveUnit.PositionDevice;

	// To Sw:
	xIclaMoving:=ABS(IclaBK.Status.iActualVelocity)>50;
	xIclaAbsMovDone:=EDGEPOS(IclaBK.Status.xInPosition);
	IF xIclaAbsMovDone THEN
		LogIclaInPosition;
	END_IF

	Block.Status.Icla.iSpeed := IclaBK.Status.iActualVelocity;
	Block.Status.Icla.xIsMoving:=IclaBK.Status.iActualVelocity<>0;

	//MOTOR   MOTOR   MOTOR   MOTOR   MOTOR   MOTOR   MOTOR   MOTOR   MOTOR   MOTOR
	//MOTOR   MOTOR   MOTOR   MOTOR   MOTOR   MOTOR   MOTOR   MOTOR   MOTOR   MOTOR
	//MOTOR   MOTOR   MOTOR   MOTOR   MOTOR   MOTOR   MOTOR   MOTOR   MOTOR   MOTOR

	MotorDriveUnit.TransmissionData:=Block.parameters.Motor.DriveUnit;

	// PowerOn Command
	AxisBK.Command.Power:= 	NOT Block.Al.xAlrSafetySystemInBlock AND
							AxisBK.Status.ControllerReady AND
							AxisBK.Status.InitDone;

	// In (mm *10)
	IF AxisBK.Status.HomeOK THEN MotorDriveUnit.pulsesDevice := AxisBK.Status.ActPosition; END_IF //TODO: Remove the HomeOK condition. Now to avoid the NotANumer error
	MotorDriveUnit.Calculation := CALC_POS_MM;
	MotorDriveUnit();
	rMotorCurrentPos:=MotorDriveUnit.PositionDevice;
	Block.Status.rMotorPosition:=rMotorCurrentPos; //Use internal var to assign it

	//Log the Position after to be in position
	IF EDGEPOS(AxisBK.Status.InPosition) THEN
		LogVertInPosition;
	END_IF

	// Position for absolute movement order	// In (mm *10)
	// Move Absolute
	MotorDriveUnit.PositionDesired := rMotorAbsPosDesired;
	MotorDriveUnit.Calculation := CALC_POS_PULSES;
	MotorDriveUnit();
	AxisBK.Parameter.Position:= MotorDriveUnit.pulsesPositionDesired;

	// Auto Acceleration, Velocity Movements
	MotorDriveUnit.AccelerationDesired := Block.parameters.Motor.rAcceleration;
	MotorDriveUnit.Calculation := CALC_ACC_PULSES;
	MotorDriveUnit();
	AxisBK.Parameter.Acceleration := MotorDriveUnit.pulsesAccelerationDesired;

	MotorDriveUnit.DecelerationDesired := Block.parameters.Motor.rDeceleration;
	MotorDriveUnit.Calculation := CALC_DEC_PULSES;
	MotorDriveUnit();
	AxisBK.Parameter.Deceleration := MotorDriveUnit.pulsesDecelerationDesired;

	//Change manual Speed
	IF xChangeMotorSpeedUp OR xChangeMotorSpeedDown THEN
		MotorDriveUnit.JogSpeedDesired := 2.0;
	ELSE
		MotorDriveUnit.JogSpeedDesired := Block.parameters.Motor.rDriveManSpeed;
	END_IF

	MotorDriveUnit.Calculation := CALC_JOGSPEED_PULSES;
	MotorDriveUnit();
	AxisBK.Parameter.JogSpeed := MotorDriveUnit.pulsesJogSpeedDesired;

	// Speed parameter for auto movements
	MotorDriveUnit.SpeedDesired := Block.parameters.Motor.rDriveAutoSpeed;
	MotorDriveUnit.Calculation := CALC_SPEED_PULSES;
	MotorDriveUnit();
	AxisBK.Parameter.Speed := MotorDriveUnit.pulsesSpeedDesired;

	// Homing: Reference Position
	MotorDriveUnit.HomePositionDesired := Block.parameters.Motor.rReferencePosition;
	MotorDriveUnit.Calculation := CALC_HOMEPOS_PULSES;
	MotorDriveUnit();
	AxisBK.Parameter.HomePosition := MotorDriveUnit.pulsesHomePositionDesired ; // Transfer in parameter structure

	// Detected incoherency with Halt and MoveAbsolute order
	IF AxisBK.Command.Move.Halt THEN
		IF xMotorAbsMovOrder THEN
			xMotorAbsMovOrder:=FALSE;
			LogMotorOrderIncoherencyHaltAndMoveAbsolute;
		END_IF
	//Removed the edgepos. It is possible because Block is executed more than x2 lower than axis
	ELSIF xMotorAbsMovOrder AND AxisBK.Status.HomeOK THEN
		AxisBK.Command.Move.Absolute:= TRUE;
		xMotorAbsMovOrder := FALSE;

		// Move absolute counter
		Block.Lg.diMoveAbsCounter:= Block.Lg.diMoveAbsCounter+1;
		//xLoggingVerMovingOrder := VerMotorOrderEventLog.Status<>ELOG_STATUS_QUEUED OR VerMotorOrderEventLog.Status<>ELOG_STATUS_LOGGING;
		//IF NOT xLoggingVerMovingOrder THEN
		//	LogVertMovementOrder;
		//END_IF
	END_IF

	IF EDGEPOS(AxisBK.Command.Move.Absolute) THEN
		LogVertMovementOrder;
	END_IF

	// Home order
	AxisBK.Command.Home:= EDGEPOS(xMotorHomeOrder);

	AxisBK.Command.Reset:= ((AxisBK.Status.ErrorID<>0) OR AxisBK.Status.PLCopenState.ErrorStop) AND Block.commands.xReset;
	AxisBK.Command.ErrorAcknowledge:= ((AxisBK.Status.ErrorID<>0) AND Block.commands.xReset) OR
										(AxisBK.Status.ErrorID=6023) OR
										(AxisBK.Status.ErrorID=29216) OR
										(AxisBK.Status.ErrorID=5001) OR
										(AxisBK.Status.ErrorID=29207) ;

END_ACTION
```

#### Inputs.st
```iecst
ACTION Inputs:

	IF NOT Block.parameters.Hw.xThereIsInTraySensor THEN
		TON_TrayInSensor.IN:= NOT Block.In.xTrayOut;
		TON_TrayInSensor.PT:= Block.parameters.tiTimeWaitTrayIn;
		TON_TrayInSensor();
		Block.In.xTrayIn := TON_TrayInSensor.Q;
	END_IF

	//Block's temperature and humidity
	Block.Status.iTemperature :=  REAL_TO_INT((Block.In.iTemperatureRaw/327.67)-40);
	Block.Status.iHumidity :=  REAL_TO_INT(Block.In.iHumidityRaw/327.67);

END_ACTION
```

#### ManualLogic.st
```iecst
ACTION ManualMovements:

	IF Block.commands.xIclaHomeOrder OR Block.commands.xBarHomeOrder OR Block.commands.xReset THEN
		RETURN;
	END_IF

	// Excessive Motor block activated
	TON_excessiveBlockActivated.IN:= (Block.commands.Mode.xManual) AND
									(AxisBK.Command.Jog.ContinuousPos OR
									AxisBK.Command.Jog.ContinuousNeg OR
									Block.commands.Manual.xManBarsUp OR
									Block.commands.Manual.xManBarsDown );
	TON_excessiveBlockActivated.PT:= T#500MS;
	TON_excessiveBlockActivated();
	xStoppedByExcessiveTimeActive:=TON_excessiveBlockActivated.Q;

	IF xStoppedByExcessiveTimeActive OR EDGEPOS(xChangeMotorSpeedUp) OR EDGEPOS(xChangeMotorSpeedDown) THEN
		Block.commands.Manual.xManBarsUp := FALSE;
		Block.commands.Manual.xManBarsDown := FALSE;
	END_IF

	// Excessive Icla activated
	TON_StoppedIclaByTimeActive.IN:= (Block.commands.Mode.xManual) AND
									(IclaBK.Command.JogBackward OR
									IclaBK.Command.JogForward OR
									Block.commands.Manual.xManIclaBack OR
									Block.commands.Manual.xManIclaForward);
	TON_StoppedIclaByTimeActive.PT:= T#3s;
	TON_StoppedIclaByTimeActive();
	xStoppedIclaByTimeActive:=TON_StoppedIclaByTimeActive.Q;
	IF xStoppedIclaByTimeActive THEN
		Block.commands.Manual.xManIclaBack := FALSE;
		Block.commands.Manual.xManIclaForward := FALSE;
	END_IF

	// Enable Up and Down movements if AnyBarEnabled
	IF NOT xStoppedByExcessiveTimeActive THEN

		Block.Status.Motor.xEnableUp:= 	((Block.commands.Mode.xManual) AND NOT Block.Status.Motor.xBarsHomed) OR //Silvia: conditions for moving when the motor is not homed (issue 1283).
										(Block.Status.Motor.xBarsHomed AND (rMotorCurrentPos<=Block.parameters.Motor.rSafePosition)); // Lower than max is allowing to go up

		Block.Status.Motor.xEnableDown:= (Block.In.xTrayIn AND Block.In.xIclaSensor AND Block.Status.Motor.xBarsHomed AND (rMotorCurrentPos>Block.parameters.Motor.rDripBarsPosition) ) OR // <357 mm position max on venturi
										( (Block.In.xTrayIn OR Block.In.xTrayOut) AND NOT Block.In.xIclaSensor AND Block.Status.Motor.xBarsHomed AND (rMotorCurrentPos>Block.parameters.Motor.rSafePositionCleanCarrier)) OR // 335.5 mm position max on venturi
										(Block.In.xTrayOut AND Block.In.xIclaSensor AND Block.Status.Motor.xBarsHomed AND rMotorCurrentPos> Block.parameters.Motor.rMinSafePosition) OR
										(NOT Block.Status.Motor.xBarsHomed AND Block.In.xTrayOut AND Block.In.xIclaSensor AND (NOT Block.Al.xAlrReferenceIncoherence AND Block.In.xReferenceDI)); //Silvia: issue 1283: we cannot move bars with the sensor broken.
	ELSE
		Block.Status.Motor.xEnableUp:=FALSE;
		Block.Status.Motor.xEnableDown:=FALSE;
	END_IF;

	////////////////
	// Block Motor
	////////////////

	// Moving up
	AxisBK.Command.Jog.ContinuousPos:= Block.Status.Motor.xEnableUp AND Block.commands.Manual.xManBarsUp AND NOT Block.commands.Manual.xManBarsDown;

	// Moving down
	AxisBK.Command.Jog.ContinuousNeg:= Block.Status.Motor.xEnableDown AND Block.commands.Manual.xManBarsDown AND NOT Block.commands.Manual.xManBarsUp;

	// Change vel.
	ManualSpeedControl;

	////////////////
	// Clean Motor
	////////////////

	// Moving forward
	IclaBK.Command.JogForward := Block.commands.Manual.xManIclaForward AND
								(Block.Status.Icla.rCurrentPosition<Block.parameters.Icla.rPositionCleanMotorFwd-2.0) AND
								(rMotorCurrentPos >= rSafeBarPosToCarrier)AND
								NOT Block.commands.Manual.xManIclaBack;
	// Moving backward
	IclaBK.Command.JogBackward:= Block.commands.Manual.xManIclaBack AND
								NOT Block.In.xIclaSensor
								AND NOT Block.commands.Manual.xManIclaForward;

	//////////////////
	// Tray Movements
	//////////////////
	IF Block.Status.PositionState <> BLOCKP_GOING_TO_PRINT AND Block.Status.PositionState <> BLOCKP_GOING_TO_CLEAN THEN
		//If in Manual the block is doing auto movements, allow them
		Block.Out.xTrayOut:= Block.commands.Manual.xManTrayOut AND ((Block.Status.Motor.xBarsHomed AND rMotorCurrentPos> Block.parameters.Motor.rDripBarsPosition) OR
																	NOT Block.Status.Motor.xBarsHomed);
		Block.Out.xTrayIn:= Block.commands.Manual.xManTrayIn AND Block.Status.Motor.xBarsHomed AND rMotorCurrentPos> Block.parameters.Motor.rDripBarsPosition;
	END_IF

	// Reset commnads as commandBoolEdge
	IF Block.commands.Manual.xManTrayOut AND Block.In.xTrayOut THEN
		Block.commands.Manual.xManTrayOut:= FALSE;
	END_IF

	IF Block.commands.Manual.xManTrayIn AND Block.In.xTrayIn THEN
		Block.commands.Manual.xManTrayIn:= FALSE;
	END_IF

	/////////////////
	// Cleaning Water Pump
	////////////////
	TP_WaterSpurtDesactDelay.IN := Block.commands.Manual.xManWaterSpurt AND Block.Status.xIsWaterBlock AND Block.In.xWaterLevelSensor;
	Block.commands.Manual.xManWaterSpurt:= FALSE; // Reset command afeter using it in the TP function
	TP_WaterSpurtDesactDelay.PT := T#2s;
	TP_WaterSpurtDesactDelay();

	Block.Out.xCleaningWaterPump := TP_WaterSpurtDesactDelay.Q;

	/////////////////
	// Capping water Pump
	////////////////
	TP_CappingWaterPumpDesactDelay.IN := Block.commands.Manual.xManCappingWaterPump AND Block.Status.xIsWaterBlock AND Block.In.xWaterLevelSensor;
	Block.commands.Manual.xManCappingWaterPump:= FALSE; // Reset command afeter using it in the TP function
	TP_CappingWaterPumpDesactDelay.PT := T#2s;
	TP_CappingWaterPumpDesactDelay();

	Block.Out.xCappingWaterPump:=TP_CappingWaterPumpDesactDelay.Q;

	/////////////////
	// Waste water Pump
	////////////////
	Tp_ManWastePump.IN := Block.commands.Manual.xManWastePump AND Block.parameters.xWastedInkTankProcess;
	Block.commands.Manual.xManWastePump:= FALSE; // Reset command afeter using it in the TP function
	Tp_ManWastePump.PT := T#2s;
	Tp_ManWastePump();

	Block.Out.xWastedInkTankPump:=Tp_ManWastePump.Q;

	////////////////////////////////
	// Enable venturi in manual state.
	Block.Out.xVenturi:= Block.commands.Manual.xManVenturi;

	//Go to Undefined if any movement is raised during Manual
	iReasonMovingMan.0 := AxisBK.Command.Jog.ContinuousPos;
	iReasonMovingMan.1 := AxisBK.Command.Jog.ContinuousNeg;
	iReasonMovingMan.2 := IclaBK.Command.JogForward;
	iReasonMovingMan.3 := IclaBK.Command.JogBackward;
	iReasonMovingMan.4 := Block.Out.xTrayOut AND NOT (Block.Status.PositionState = BLOCKP_GOING_TO_PRINT OR Block.Status.PositionState = BLOCKP_GOING_TO_CLEAN);
	iReasonMovingMan.5 := Block.Out.xTrayIn AND NOT (Block.Status.PositionState = BLOCKP_GOING_TO_PRINT OR Block.Status.PositionState = BLOCKP_GOING_TO_CLEAN);
	IF iReasonMovingMan >0 THEN
		Block.Status.PositionState := BLOCKP_UNDEFINED;
	END_IF

	//First Home direct to enable movement of the drive
	IF 	NOT AxisBK.Status.HomeOK AND NOT Block.Status.Motor.xBarsHoming THEN
		//AxisBK.Parameter.HomePosition:=AxisBK.Status.ActPosition;
		AxisBK.Command.HomeDirect:=TRUE;
	END_IF

END_ACTION

ACTION HomingIcla:

	IF xBlockPosChange THEN
		Block.commands.xIclaHomeOrderInterrupt:=FALSE;
		nState := 110;
	END_IF

	CASE nState OF

		(*----------------------------------- ICLA HOMING ----------------------------------------------------------*)
		(*----------------------------------- ICLA HOMING ----------------------------------------------------------*)
		(*----------------------------------- ICLA HOMING ----------------------------------------------------------*)

		110:
			iLastState:=nState;
			// Homing Reference before movements to asure that Icla is refrenced
			Block.Status.Icla.xHomed :=FALSE;
			IF NOT IclaBK.Status.xReferenced THEN
				//It is a Home Direct adn doesnt need wait for nothing
				// IclaBK.Status.xReferenced is done when home ok
				//In CASE first connection OF the Icla TO the machine. Internally it is NOT homed
				IclaBK.Command.Home:= TRUE;
			ELSE
				nState:= nState+1;	 // Finished actions for order reference Icla before any movement
			END_IF

		111:
			// If Icla In Sensor, go out
			iLastState:=nState;
			IF Block.In.xIclaSensor THEN
				nState:= nState+1;		//Going to forward movement
			ELSE
				nState:= nState+2; 		//Going to backward movement
			END_IF

		112:
			//Starting forward movement IN ABSOLUTE
			iLastState:=nState;
			IclaBK.Command.JogForward:=TRUE;
			//Stop movement when not IclaIndSensor
			IF NOT Block.In.xIclaSensor THEN
				IclaBK.Command.JogForward:=FALSE;
				nState:= nState+1;
			END_IF

		113:
			iLastState:=nState;
			//Starting backward movement when the Icla is stopped
			IF NOT Block.Status.Icla.xIsMoving THEN
				IclaBK.Command.JogBackward:=TRUE;
				nState:= nState+1;
			END_IF

		114:
			iLastState:=nState;
			// Gone back to sensor and when it arrived we have to stop movements as mandatory
			IF Block.In.xIclaSensor THEN
				IclaBK.Command.JogBackward:=FALSE;
				nState:= nState+1;
			END_IF

		115:
			iLastState:=nState;
			// Homing Done, with double check of cleaning carriage sensor
			IF NOT Block.Status.Icla.xIsMoving THEN
				nState:= nState+1;
			END_IF

		116:
			iLastState:=nState;
			// Homing Done, with double check of cleaning carriage sensor
			IclaBK.Command.Home:= TRUE;
			IF (IclaBK.Status.xReferenced) THEN
				// Homing Done, with double check of cleaning carriage sensor
				Block.commands.xIclaHomeOrder:=FALSE;
				Block.Status.Icla.xHomed :=TRUE;
				nState:= 0;
				// Finished actions for order homing
			END_IF

	END_CASE

END_ACTION

ACTION HomingBar:

	IF xBlockPosChange THEN
		AxisBK.Command.QuickStop:=FALSE;				// Reset state QuickStop
		nState := 150;
	END_IF

	CASE nState OF

		(*----------------------------------- BAR HOMING ----------------------------------------------------------*)
		(*----------------------------------- BAR HOMING ----------------------------------------------------------*)
		(*----------------------------------- BAR HOMING ----------------------------------------------------------*)

		150:
			iLastState:=nState;
			Block.Status.Motor.xBarsHomed:= FALSE;
			AxisBK.Status.HomeOK := FALSE;
			xMotorHomeOrder:= TRUE;
			nState:=nState+1;

		151:
			iLastState:=nState;
			IF AxisBK.Status.HomeOK THEN
				xMotorHomeOrder:= FALSE;
				Block.commands.xBarHomeOrder:=FALSE;
				Block.Status.Motor.xBarsHomed:= TRUE;
				nState:= 0;
			END_IF

	END_CASE

END_ACTION

ACTION GoingToClean:

	IF xBlockPosChange THEN
		AxisBK.Command.QuickStop:=FALSE;				// Reset state QuickStop
		nState := 190;
	END_IF

	CASE nState OF

		(*----------------------------------- GOING TO CLEAN ------------------------------------------------------*)
		(*----------------------------------- GOING TO CLEAN ------------------------------------------------------*)
		(*----------------------------------- GOING TO CLEAN ------------------------------------------------------*)

		190:
			iLastState:=nState;

			ResetKnownPositions;

			MoveBarsToCleanPosition;

		191:
			iLastState:=nState;

			CheckAbsolutMovementFinished;

		192:
			iLastState:=nState;
			xInClean:= TRUE;
			nState:= 0;

	END_CASE

END_ACTION

ACTION ManualSpeedControl:

	IF NOT Block.Status.Motor.xBarsHomed THEN
		xChangeMotorSpeedUp		:= FALSE;
		xChangeMotorSpeedDown	:= FALSE;
		RETURN;
	END_IF

	IF AxisBK.Command.Jog.ContinuousNeg THEN //DOWN

		xChangeMotorSpeedUp := FALSE;

		IF  (rMotorCurrentPos <= Block.parameters.Motor.rDripBarsPosition + Block.parameters.Motor.rReduceSpeedDistance AND Block.In.xTrayIn) OR
			(rMotorCurrentPos <= Block.parameters.Motor.rSafePositionCleanCarrier + Block.parameters.Motor.rReduceSpeedDistance AND NOT Block.In.xIclaSensor) OR
			rMotorCurrentPos <= Block.parameters.Motor.rMinSafePosition + Block.parameters.Motor.rReduceSpeedDistance THEN

			xChangeMotorSpeedDown := TRUE;

		END_IF

	ELSIF AxisBK.Command.Jog.ContinuousPos THEN //UP

		xChangeMotorSpeedDown := FALSE;

		IF rMotorCurrentPos >= Block.parameters.Motor.rSafePosition - Block.parameters.Motor.rReduceSpeedDistance THEN

			xChangeMotorSpeedUp := TRUE;

		END_IF

	ELSIF NOT ((rMotorCurrentPos <= Block.parameters.Motor.rDripBarsPosition + Block.parameters.Motor.rReduceSpeedDistance OR
		rMotorCurrentPos <= Block.parameters.Motor.rSafePositionCleanCarrier + Block.parameters.Motor.rReduceSpeedDistance OR
		rMotorCurrentPos <= Block.parameters.Motor.rMinThicknessMedia + Block.parameters.Motor.rReduceSpeedDistance) OR
		(rMotorCurrentPos >= Block.parameters.Motor.rSafePosition - Block.parameters.Motor.rReduceSpeedDistance)) THEN

		xChangeMotorSpeedUp		:= FALSE;
		xChangeMotorSpeedDown	:= FALSE;

	END_IF

END_ACTION
```

#### ValvesUnit.st
```iecst
ACTION ValvesUnit:

	//If comms is not CanOpen, just go out
	IF Block.parameters.Hw.ValvesCommsType <> COMMS_CANOPEN THEN
		RETURN;
	END_IF

	CanGetState.enable := TRUE;
	CanGetState.node := Block.parameters.Hw.ValvesNode;
	CanGetState.pDevice := ADR('IF7');
	CanGetState();

	iReasonNotValveComms.0 := CanGetState.state = coPREOPERATIONAL;
	iReasonNotValveComms.1 := CanGetState.state = coUNKNOWN;
	iReasonNotValveComms.2 := CanGetState.state = coNOTAVAIL;

	tonNotValveComms.IN := iReasonNotValveComms > 0;
	tonNotValveComms.PT := t#3s;
	tonNotValveComms();

	xChangedValvesState := ValvesCanResetState_copy <> ValvesCanResetState;
	ValvesCanResetState_copy := ValvesCanResetState;

	CASE ValvesCanResetState OF

		COCOMSR_UNDEFINED,
		COCOMSR_COMMUNICATING:

			iTimesTryToReset := 0;

			//If time in error, define an error comms
			IF tonNotValveComms.Q THEN
				ValvesCanResetState := COCOMSR_COMMSERROR;
			END_IF

		COCOMSR_COMMSERROR:

			//Start the resetting process
			IF Block.commands.xReset THEN
				ValvesCanResetState := COCOMSR_RESETTING;
			END_IF

			//Communication has returned to work
			IF CanGetState.state = coOPERATIONAL THEN
				ValvesCanResetState := COCOMSR_COMMUNICATING;
			END_IF

		COCOMSR_RESETTING:

			CANopenResetValves.enable := TRUE;
			CANopenResetValves.node := Block.parameters.Hw.ValvesNode;
			CANopenResetValves.pDevice := ADR('IF7');
			CANopenResetValves.state := coRESET_NODE;
			CANopenResetValves();

			IF CANopenResetValves.status = ERR_OK THEN
				lastCanOpenResetError := CANopenResetValves.error;
				CANopenResetValves(enable := FALSE);
				ValvesCanResetState := COCOMSR_WAITINGTOBERESETTED;
			END_IF

			tonValveCommsErrorResetting.IN := NOT xChangedValvesState;
			tonValveCommsErrorResetting.PT := t#10s;
			tonValveCommsErrorResetting();

			IF tonValveCommsErrorResetting.Q THEN
				lastResetingState := CanGetState.state;
				lastFbResetStatus := CANopenResetValves.status;
				tonValveCommsErrorResetting(IN:=FALSE);
				CANopenResetValves(enable:=FALSE);
				ValvesCanResetState := COCOMSR_RESETTING_ERROR;
			END_IF

		COCOMSR_WAITINGTOBERESETTED:

			//Communication has returned to work
			IF CanGetState.state = coOPERATIONAL THEN
				ValvesCanResetState := COCOMSR_COMMUNICATING;
			END_IF

			tonValveCommsErrorResetting.IN := NOT xChangedValvesState;
			tonValveCommsErrorResetting.PT := t#4s;
			tonValveCommsErrorResetting();

			IF tonValveCommsErrorResetting.Q THEN
				lastResetingState := CanGetState.state;
				lastFbResetStatus := CANopenResetValves.status;
				tonValveCommsErrorResetting(IN:=FALSE);
				ValvesCanResetState := COCOMSR_RESETTING_ERROR;
			END_IF

		COCOMSR_RESETTING_ERROR:

			//After an error, wait to try again
			tonValveCommsErrorResetting.IN := NOT xChangedValvesState;
			tonValveCommsErrorResetting.PT := t#500ms;
			tonValveCommsErrorResetting();

			IF tonValveCommsErrorResetting.Q  AND iTimesTryToReset < 6 THEN
				iTimesTryToReset := iTimesTryToReset + 1;
				ValvesCanResetState := COCOMSR_RESETTING;
			ELSIF tonValveCommsErrorResetting.Q THEN
				ValvesCanResetState := COCOMSR_COMMSERROR;
			END_IF

	END_CASE

END_ACTION
```

### Program Logical/ExtPack/BlockCtrl/BlockCtrl_v1/InitBlockCtrl

#### InitiBlock.st
```iecst
PROGRAM _CYCLIC
	gIndexBlock:= 1;
END_PROGRAM
```

### Program Logical/ExtPack/BlockCtrl/BlockSim/BlockSim_v1/BlockSim (IEC)

#### Main.st - Init, cyclic, exit code
```iecst
PROGRAM _CYCLIC
	(* Insert code here *)

	Block ACCESS ADR(gBlock[iBlockSimIndex]);
	MotorBlock  ACCESS ADR (gAxis[Block.parameters.iMotorAxisIndex]);
	IclaBK ACCESS ADR (gIcla[Block.parameters.iIclaAxisIndex]);
	SimBlock ACCESS ADR (gSimBlock[iBlockSimIndex]);

	//If the motor is not defined, it is considered there is no real block and return to avoid attach null pointer
	IF Block.parameters.iMotorAxisIndex = 0 THEN
		iBlockSimIndex:= iBlockSimIndex + 1;
		RETURN;
	END_IF

	//Enabling homing the icla
	IF Block.Status.Icla.xHomed THEN
		Block.In.xIclaSensor:=IclaBK.Status.iActualPosition<=0;
	END_IF

	//Automate referencing the sensor
	IF Block.Status.iBlockCaseLogicControl = 112 THEN
		Block.In.xIclaSensor:=FALSE;
	END_IF
	IF Block.Status.iBlockCaseLogicControl = 114  AND NOT SimBlock.Commands.DelayHomingIcla THEN
		Block.In.xIclaSensor:=TRUE;
	END_IF

	//Managing the Sensor signal with the position of hte Icla
	IF Block.commands.Mode.xAuto THEN
		Block.In.xIclaSensor:=IclaBK.Status.iActualPosition<=0;
	END_IF

	//Capping flow meter sensor
	IF Block.parameters.xCappingProcess THEN
		Block.In.xCappingWaterFlowmeter := TRUE;
	ELSE
		Block.In.xCappingWaterFlowmeter := FALSE;
	END_IF

	//Managing the homing of the Elevation motor
	IF EDGEPOS(MotorBlock.Status.PLCopenState.Homing AND NOT SimBlock.Commands.DelayHomingBar ) THEN
		iRefSignalState:=1;
		TimesExcecHoming:=TimesExcecHoming+1;
	END_IF

	StatusNcAccess := ncaccess(ncACP10MAN, ADR(MotorBlock.Parameter.Init.AxisObjectName), ADR(AxisRef));

	fbWriteRefSignal.Axis := AxisRef;
	fbWriteRefSignal.ParID := ACP10PAR_VAR_I4_0;
	fbWriteRefSignal.DataType := ncPAR_TYP_DINT;
	fbWriteRefSignal.DataAddress := ADR(uiValueRef);

	CASE iRefSignalState OF
		0:
			fbWriteRefSignal.Execute := FALSE;
		1:
			//IF EDGEPOS(iRefSignalState=2) THEN fbWriteRefSignal.Execute := TRUE; END_IF
			IF NOT fbWriteRefSignal.Done AND NOT fbWriteRefSignal.Busy THEN
				fbWriteRefSignal.Execute := TRUE;
			END_IF
			uiValueRef:=1;
			IF fbWriteRefSignal.Done THEN
				fbWriteRefSignal.Execute := FALSE;
				iRefSignalState:=2;
			END_IF
			IF fbWriteRefSignal.Error THEN
				fbWriteRefSignal.Execute := FALSE;
			END_IF

		2:
			//IF EDGEPOS(iRefSignalState=2) THEN fbWriteRefSignal.Execute := TRUE; END_IF
			IF NOT fbWriteRefSignal.Done AND NOT fbWriteRefSignal.Busy THEN
				fbWriteRefSignal.Execute := TRUE;
			END_IF
			uiValueRef:=0;
			IF fbWriteRefSignal.Done THEN
				fbWriteRefSignal.Execute := FALSE;
				iRefSignalState:=3;
			END_IF

		3:
			//IF EDGEPOS(iRefSignalState=2) THEN fbWriteRefSignal.Execute := TRUE; END_IF
			IF NOT fbWriteRefSignal.Done AND NOT fbWriteRefSignal.Busy THEN
				fbWriteRefSignal.Execute := TRUE;
			END_IF
			uiValueRef:=1;
			IF fbWriteRefSignal.Done THEN
				fbWriteRefSignal.Execute := FALSE;
				iRefSignalState:=0;
			END_IF

	END_CASE

	fbWriteRefSignal();

	iBlockSimIndex:= iBlockSimIndex + 1;

END_PROGRAM
```

#### BlockSim.var - Local variables
```iecst
VAR
	Block : REFERENCE TO StBlock;
	MotorBlock : REFERENCE TO AxisCtrl_typ;
	IclaBK : REFERENCE TO stIcla;
	SimBlock : REFERENCE TO SimBlock_typ;
	fbWriteRefSignal : MC_BR_WriteParID;
	iRefSignalState : USINT;
	AxisRef : UDINT;
	StatusNcAccess : UINT;
	uiValueRef : DINT;
	TimesExcecHoming : USINT;
END_VAR
```

- Program Logical/ExtPack/BlockCtrl/BlockSim/BlockSim_v1/InitBlockSim (IEC) (no source held here)

### SimpleBlockCtrl.typ
```iecst
TYPE
	SimpleBlock_Outputs : 	STRUCT
		xEnableDrive : BOOL;
	END_STRUCT;
	SimpleBlock_Log : 	STRUCT
		diMoveARelCounter : DINT;
		diMoveAbsCounter : DINT;
		diHomingsNumber : DINT;
	END_STRUCT;
	SimpleBlock_Alarms : 	STRUCT
		xAlrSafetySystemInBlock : BOOL; (*CriticalAlarm*)
		xAlrReferenceIncoherence : BOOL; (*CriticalAlarm*)
		xAlrDriveProtection : BOOL; (*CriticalAlarm*)
		xAlrBarMtrNoRef : BOOL; (*CriticalAlarm *)
		xAlrComBarMtr : BOOL; (*CriticalAlarm *)
		xAnyDriveAlarm : BOOL; (*CriticalAlarm *)
		xAlBarMotorPowerOff : BOOL;
		xAlrBlockReachedMaxPosition : BOOL;
		xBarMotorTemp : BOOL; (*Warning: Bar Motor Temperature Too Hot*)
		xBarDriverTemp : BOOL; (*Warning: Bar Driver Temperature Too Hot*)
		xAlrCheckHomingSensor : BOOL; (*Warning: Bar Homing Sensor Maybe Broken*)
		xAlrEmergencyStop : BOOL; (*Emergency button pushed without diferenciating front or rear*)
	END_STRUCT;
	SimpleBlock_commandsManual : 	STRUCT
		xManBarsUp : BOOL; (*Command just in manual mode*)
		xManBarsDown : BOOL; (*Command just in manual mode*)
	END_STRUCT;
	SimpleBlock_commands : 	STRUCT
		Mode : StGeneral_States_Mode;
		StateMode : enumEFI_GenMachineState; (*commands to block*)
		AutoMode : stEFI_MachineAutoModes; (*commands to inform belt*)
		Manual : SimpleBlock_commandsManual;
		xBarHomeOrder : BOOL; (*State Command just in manual mode*)
		xToPrint : BOOL; (*Command just in AUTO mode*)
		xToCap : BOOL; (*Command just in AUTO mode*)
		xToPrintLab : BOOL; (*EDGE Command. Reseted manually in Block*)
		xToCapLab : BOOL; (*EDGE Command. Reseted manually in Block*)
		xMute : BOOL; (*Command Bool mute sound*)
		xReset : BOOL; (*Command Bool Reset*)
	END_STRUCT;
	SimpleBlock_Parameters_Motor : 	STRUCT
		DriveUnit : MC_DriveUnitManager;
		rPrintPosition : REAL; (*Input from LC Band. Value in mm*)
		rDriveManSpeed : REAL; (*Vertical motor manual speed. Value in mm/s*)
		rDriveAutoSpeed : REAL; (*Vertical motor automatic speed. Value in mm/s*)
		rCapPosition : REAL; (*Capped position in mm*)
		rSafePosition : REAL; (*Position in mm*)
		rMinSafePosition : REAL; (*Position in mm*)
		rReferencePosition : REAL; (*Reference Position in mm*)
		rMinThicknessMedia : REAL; (*Minimum media thickness in mm*)
		VerticalDirection : MotorDirection_enum; (*To indicate that the motor must spin in reverse*)
		uiMaxCurrentBarsUp : UINT;
		uiMaxCurrentBarsDown : UINT;
		uiColisionCurrentUp : UINT;
		uiColisionCurrentDown : UINT;
		rReduceSpeedDistance : REAL; (*Distance to the limit to reduce manual speed*)
		rAcceleration : REAL;
		rDeceleration : REAL;
		xOversized : BOOL; (*Variable to define motor's operation torque is much lower than the rated torque*)
		rOperationTorque : REAL; (*Motor's operation torque*)
	END_STRUCT;
	SimpleBlock_SwParameters : 	STRUCT
		xEnableToMovements : BOOL; (*Block is enalbed to movements and doesnt go to print if order is received,  Cleaning? *)
		xEnableToPrint : BOOL; (*Block is enalbed to print and it goes to print if order is received,*)
		rOffsetPrintMotor : REAL; (*Software Input. Printer description, advanced (adjust the motor block position)*)
		rOffsetCappingMtr : REAL;
	END_STRUCT;
	SimpleBlock_Parameters_Hw : 	STRUCT
		xExistBlock : BOOL;
	END_STRUCT;
	SimpleBlock_Parameters : 	STRUCT
		Motor : SimpleBlock_Parameters_Motor;
		Hw : SimpleBlock_Parameters_Hw;
		iMotorAxisIndex : INT; (*Index of the vertical motor to assign it*)
		xBeltIsEmpty : BOOL; (*The machine send the information that the belt is empty*)
		xLeftHandMachine : BOOL; (*To indicate that the machine is left hand.*)
		xRightHandMachine : BOOL; (*To indicate that the machine is right hand.*)
	END_STRUCT;
	SimpleBlock_MotorStatus : 	STRUCT
		xBarsHomed : BOOL;
		xBarsHoming : BOOL;
		rActPosition : REAL; (*Actual Position of the motor in Motor units*)
		rIntensty : REAL; (*Intensity in Amperes (A)*)
		rSpeed : REAL; (*Actual Speed of the axis in mm/s*)
		rOperationTorque : REAL; (*Motor's operation torque*)
		rTorque : REAL; (*Actual Torque of the axis in Nm*)
		xEnableUp : BOOL;
		xEnableDown : BOOL;
		ErrorID : UINT; (*ErrorID of any occurred error*)
	END_STRUCT;
	SimpleBlock_StatusPosition : 	STRUCT
		xUndefined : BOOL;
		xInCap : BOOL;
		xInPrint : BOOL;
		xGoingToCap : BOOL;
		xGoingToPrint : BOOL;
		xReadyToPrint : BOOL; (*In print postion without safe offsets position*)
	END_STRUCT;
	SimpleBlock_Status : 	STRUCT
		iBlockCaseLogicControl : INT; (*nState logic control*)
		iBlockState : INT; (*Value to send to Sw: 0=NO_AUTO, 1=IN_CAP, 2=IN_PRINT, 3=CLEANING, 4=GOING_TO_CAP, 5=GOING_TO_PRINT*)
		xEnabledMovements : BOOL;
		xAnyManualMovement : BOOL;
		BlockState : Block_States_enum := BLOCK_STOPPING;
		PositionState : Block_Position_enum := BLOCKP_UNDEFINED;
		Position : SimpleBlock_StatusPosition;
		xCleaningDone : BOOL; (*EDGE*)
		xGoingUpWithNoConsent : BOOL;
		xEnabledToPrint : BOOL;
		xAlarmToEmptyBelt : BOOL; (*This Block has an alarm that requires to empy the belt*)
		rMotorPosition : REAL; (*To Software. Value in mm*)
		execTimes : UDINT;
		Motor : SimpleBlock_MotorStatus;
	END_STRUCT;
	SimpleBlock_Inputs : 	STRUCT
		xReferenceDI : BOOL;
		xSafetyOK : BOOL; (*Bar Safety Is Ok*)
		xVertTopLimit : BOOL;
		xDifferentialOK : BOOL;
		xDriveProtectionOK : BOOL;
		xEmergencyStop : BOOL; (*Emergency button pushed without diferenciating front or rear*)
	END_STRUCT;
	SimpleBlock : 	STRUCT
		In : SimpleBlock_Inputs;
		Status : SimpleBlock_Status;
		parameters : SimpleBlock_Parameters;
		parSw : SimpleBlock_SwParameters;
		commands : SimpleBlock_commands; (*all block commands*)
		AlSummary : stEFI_AlarmSummary;
		Al : SimpleBlock_Alarms;
		Lg : SimpleBlock_Log;
		Out : SimpleBlock_Outputs;
	END_STRUCT;
END_TYPE
```

### SimpleBlockCtrl.var
```iecst
VAR
	gIndexSimpleBlock : USINT;
END_VAR
```

- Program Logical/ExtPack/SimpleBlockCtrl/SimpleBlockCtrl_v1/InitSimpleBlockCtrl (IEC) (no source held here)

### Program Logical/ExtPack/SimpleBlockCtrl/SimpleBlockCtrl_v1/SimpleBlockCtrl

#### AlarmSound.st
```iecst
ACTION AlarmSound:

	//////////////////////////////
	// BLOCK SOUNDS
	//////////////////////////////

	// Reseteable alarms. Reset is input in the ars function
	// Alarms reseteable sound management. //TOJC: Pending check all alarms!

	ars_AlrSafetySystemInBlock.xAlarm:= Block.Al.xAlrSafetySystemInBlock AND Block.commands.StateMode<>PRINTERGEN_ZERO;
	ars_AlrSafetySystemInBlock.xSilence:= Block.commands.xMute;
	ars_AlrSafetySystemInBlock();

	ars_DriveAlarm.xAlarm:= (Block.Al.xAnyDriveAlarm AND Block.Status.Motor.xBarsHomed);
	ars_DriveAlarm.xSilence:= Block.commands.xMute;
	ars_DriveAlarm();

	ars_AlrComBarMtr.xAlarm:= Block.Al.xAlrComBarMtr;
	ars_AlrComBarMtr.xSilence:= Block.commands.xMute;
	ars_AlrComBarMtr();

	ars_BrokenReferSensor.xAlarm:= Block.Al.xAlrReferenceIncoherence;
	ars_BrokenReferSensor.xSilence:= Block.commands.xMute;
	ars_BrokenReferSensor();

	ars_EmergencyStop.xAlarm:= Block.Al.xAlrEmergencyStop;
	ars_EmergencyStop.xSilence:= Block.commands.xMute;
	ars_EmergencyStop();

	Block.AlSummary.xAlarmSound:=	ars_AlrSafetySystemInBlock.xAlarmSound OR
									ars_DriveAlarm.xAlarmSound OR
									ars_AlrComBarMtr.xAlarmSound OR
									ars_EmergencyStop.xAlarmSound OR
									(xAnyManualMov AND gPLC.xBlk_200ms);

	// Block sounds while is homing
	// Sound generation for homing process
	// Sound generation: manual movements
	xAnyManualMov:=Block.Status.Motor.xBarsHoming OR
					AxisBK.Command.Jog.ContinuousPos OR
                	AxisBK.Command.Jog.ContinuousNeg;

END_ACTION
```

#### AlarmsSummary.st
```iecst
ACTION AlarmsSummary:

	// Stop Alarms. The machine goes to Automatic-Stop.
	iReasonStop.0 := Block.Al.xAnyDriveAlarm;
	iReasonStop.1 := Block.Al.xAlrBarMtrNoRef;
	iReasonStop.2 := Block.Al.xAlrComBarMtr;

	Block.AlSummary.xAlarmStop:= iReasonStop > 0;
	IF EDGEPOS(Block.AlSummary.xAlarmStop) THEN
		Block.AlSummary.iReasonStop[0] := iReasonStop;
		LogStopAlarm;
	ELSIF EDGEPOS(NOT Block.commands.AutoMode.xStop AND NOT Block.AlSummary.xAlarmStop) THEN
		Block.AlSummary.iReasonStop[0] := 0;
	END_IF

	// Out of Automatic Alarms. The machine goes to Standby mode.
	iReasonCritical.0 := (Block.Al.xAlrSafetySystemInBlock AND Block.Status.xEnabledMovements);
	iReasonCritical.1 := Block.Al.xAlrDriveProtection;
	Block.AlSummary.xAlarmCritical:= iReasonCritical > 0;

	//Register the reason of the Critical Alarm
	IF Block.commands.Mode.xAuto AND EDGEPOS(Block.AlSummary.xAlarmCritical) THEN
		Block.AlSummary.iReasonCritical := iReasonCritical;
		LogCriticalAlarm;
	ELSIF EDGEPOS(Block.commands.Mode.xAuto AND NOT Block.AlSummary.xAlarmCritical) THEN
		Block.AlSummary.iReasonCritical := 0;
	END_IF

	// Any alarm
	Block.AlSummary.xAnyAlarm:= Block.AlSummary.xAlarmStop OR Block.AlSummary.xAlarmCritical;

	// Warning alarms (used in AlarmaAvisoExterno)
	iReasonAnyWarning.5 := Block.Al.xBarDriverTemp;
	iReasonAnyWarning.6 := Block.Al.xBarMotorTemp;
	iReasonAnyWarning.7 := Block.Al.xAlrCheckHomingSensor;
	iReasonAnyWarning.8 := Block.Al.xAlrBlockReachedMaxPosition;
	iReasonAnyWarning.13 := Block.Al.xAlrReferenceIncoherence;
	Block.AlSummary.xAnyWarning:= iReasonAnyWarning > 0 ;

	//Alarm Safety System General
	iReasonSafetyGeneral.1 := Block.Al.xAlrSafetySystemInBlock;
	Block.AlSummary.xAlrSafetySystemGeneral:= iReasonSafetyGeneral > 0;

END_ACTION
```

#### AutoLogic.st
```iecst
ACTION GoingToCap:

	IF xBlockPosChange THEN
		nState := 208;
	END_IF

	CASE nState OF

		(*STOP POSITION     --------------------------------------------------------*)
		(*STOP POSITION     --------------------------------------------------------*)
		(*STOP POSITION     --------------------------------------------------------*)

		208:
			iLastState:=nState;
			ResetKnownPositions;
			nState:= nState+1;

		209:
			iLastState:=nState;
			IF AxisBK.Status.ErrorID=0 THEN
				StopMovements;
				nState:= nState+1;
			END_IF

		210:
			iLastState:=nState;
			IF AllDevicedStopped(ADR(Block), ADR(AxisBK)) THEN
				IF AxisBK.Status.PowerOn  AND AxisBK.Status.PLCopenState.StandStill THEN
					nState:= nState+1;
				END_IF
			END_IF

		211:
			iLastState:=nState;

			// If It is in safe place we go to next step
			IF ABS(rMotorCurrentPos-Block.parameters.Motor.rCapPosition)<0.01 THEN
				nState:= nState+3;
			ELSE
				nState:= nState+1;
			END_IF

			// Here Alarm risk colision when Icarriage is not in sensor?

		212:
			iLastState:=nState;
			MoveBarsToCapPosition; //Directly nState:= nState+1;

		213:
			iLastState:=nState;
			CheckAbsolutMovementFinished; //If Finished, nState:= nState+1;

		214:
			iLastState:=nState;
			xInCap:= TRUE;
			nState:= 0;

	END_CASE

END_ACTION

ACTION GoingToPrint:

	IF xBlockPosChange THEN
		nState := 217;
	END_IF

	CASE nState OF

		(*PRINT POSITION    --------------------------------------------------------*)
		(*PRINT POSITION    --------------------------------------------------------*)
		(*PRINT POSITION    --------------------------------------------------------*)

		217:
			iLastState:=nState;

			ResetKnownPositions;

			nState:= nState+1;

		218:
			iLastState:=nState;
			IF AxisBK.Status.ErrorID=0 THEN
				StopMovements;
				nState:= nState+1;
			END_IF

		219:
			iLastState:=nState;
			IF AllDevicedStopped(ADR(Block), ADR(AxisBK)) THEN
				IF AxisBK.Status.PowerOn AND AxisBK.Status.PLCopenState.StandStill THEN
					nState:= nState+1;
				END_IF
			END_IF

		220:
			iLastState:=nState;
			//Going to print
			rMotorAbsPosDesired:= rCalcPosDesPrint;
			xMotorAbsMovOrder:= TRUE;

			nState:= nState+1;

		221:
			iLastState:=nState;

			IF ABS(rMotorCurrentPos-rMotorAbsPosDesired)<0.01 THEN
				xInPrint:= TRUE;
				nState:= 0;
			END_IF

	END_CASE

END_ACTION

ACTION MoveBarsToCapPosition:
	//Created an action because this code is called from 2 different places
	rMotorAbsPosDesired:= Block.parameters.Motor.rCapPosition;
	xMotorAbsMovOrder:= TRUE;
	nState:= nState+1;

END_ACTION

ACTION CheckAbsolutMovementFinished:

	IF ABS(rMotorCurrentPos-rMotorAbsPosDesired)<0.01 THEN
		nState:= nState+1;
	END_IF

END_ACTION
```

#### BlockManager.st
```iecst
PROGRAM _CYCLIC

	// Block Reference
	Block ACCESS ADR(gSimpleBlock[gIndexSimpleBlock]);
	AxisBK ACCESS ADR (gAxis[Block.parameters.iMotorAxisIndex]);

	//If the Block doesn't exist, remove alarms and exit. Extra condition to avoid a divided by 0 error at start
	IF NOT Block.parameters.Hw.xExistBlock THEN
		ResetAlarms;
		gIndexSimpleBlock := gIndexSimpleBlock + 1;
		RETURN;
	END_IF

	//Limit the value of parameters configured
	BlockParameters;

	IF Block.parSw.xEnableToMovements THEN
		Block.Status.xEnabledMovements:= TRUE;
	ELSIF NOT Block.parSw.xEnableToMovements AND (xInCap OR NOT Block.Status.Motor.xBarsHomed) THEN
		Block.Status.xEnabledMovements:= FALSE;
	END_IF

	IF Block.commands.xReset THEN
		ResetAlarms;
	END_IF

	BlockAlarms;
	AlarmSound;

	IF (NOT Block.Status.xEnabledMovements) THEN
		gIndexSimpleBlock := gIndexSimpleBlock + 1;
		RETURN;
	END_IF

	ControlState;

	BlockStatesCtrl;

	InputParamsMotors;

	ResetEdgeCommands;

	//Increased exec times number to be checked outside
	Block.Status.execTimes := Block.Status.execTimes + 1;

	// Index added
	gIndexSimpleBlock := gIndexSimpleBlock + 1;

END_PROGRAM
```

#### BlockParameters.st
```iecst
ACTION BlockParameters:

	// Print motor offset
	Block.parSw.rOffsetPrintMotor		:= MAX(Block.parSw.rOffsetPrintMotor,GC_MIN_OFFSET_BLOCK);

	//Assign the direction of the vertical motor
	IF Block.parameters.Motor.VerticalDirection=MOTOR_NEGATIVE THEN
		AxisBK.Parameter.Direction:=MOTOR_NEGATIVE_AXIS;
	ELSE
		AxisBK.Parameter.Direction:=MOTOR_POSITIVE_AXIS;
	END_IF

END_ACTION
```

#### BlockStateGen.st
```iecst
ACTION BlockStateGen:

	// PRINT POSITION ORDER
	xOrderToPrint:=	(Block.commands.xToPrint AND Block.parSw.xEnableToPrint) OR
					(Block.commands.xToPrintLab AND Block.commands.AutoMode.xLaboratory);

	// CAP POSITION ORDER
	xCapOrder:= Block.commands.xToCap OR
				(Block.commands.xToCapLab AND Block.commands.AutoMode.xLaboratory) OR
				EDGENEG(Block.parSw.xEnableToPrint);

	CASE Block.Status.BlockState OF

		BLOCK_STOPPED:
			AxisBK.Command.QuickStop:=FALSE;

		BLOCK_STOPPING:
			StopMovements;
			IF AllDevicedStopped(ADR(Block), ADR(AxisBK)) THEN
				Block.Status.BlockState := BLOCK_STOPPED;
			END_IF

		BLOCK_MANUAL:
			ManualMovements;

			// To do home in block is mandatory to have Icla at sensor and try out
			IF Block.commands.xBarHomeOrder THEN

				Block.Status.PositionState := BLOCKP_HOMING_BAR;

			END_IF

		BLOCK_AUTO:

			IF (xCapOrder AND NOT xInCap AND Block.Status.Motor.xBarsHomed) THEN
				//I movoe to STOP
				Block.Status.PositionState := BLOCKP_GOING_TO_CAP;

			ELSIF xOrderToPrint AND NOT xInPrint AND NOT Block.AlSummary.xAlarmCritical AND NOT Block.AlSummary.xAlarmStop THEN
				//Going TO PRINT
				Block.Status.PositionState := BLOCKP_GOING_TO_PRINT;

			END_IF

	END_CASE

END_ACTION
```

#### BlockStateMach.st
```iecst
ACTION BlockStateMach:

	CASE Block.commands.StateMode OF

		PRINTERGEN_ZERO:
			//When entering in Zero, go to Stopping
			IF MachineStatePrevious<>PRINTERGEN_ZERO THEN
				Block.Status.BlockState := BLOCK_STOPPING;
				//If the block is not in a clear position, go to undefined
				IF Block.Status.PositionState = BLOCKP_GOING_TO_CAP OR
					Block.Status.PositionState = BLOCKP_GOING_TO_PRINT 	THEN

					Block.Status.PositionState := BLOCKP_UNDEFINED;

				END_IF
				nState :=0;
			END_IF

		PRINTERGEN_MANUAL:
			IF Block.Status.BlockState = BLOCK_STOPPED THEN
				Block.Status.BlockState := BLOCK_MANUAL;
			END_IF

		PRINTERGEN_AUTO:
			IF Block.Status.BlockState = BLOCK_STOPPED THEN
				Block.Status.BlockState := BLOCK_AUTO;
			END_IF

	END_CASE

END_ACTION
```

#### BlockStatesCtrl.st
```iecst
ACTION BlockStatesCtrl:

	//Desired print position is max value because rPrintPosition comes form belt algorithm corecction based on matrix at LC_Band.st. It gives rPrintPosition calculated by matrix
	rCalcPosDesPrint:= MAX (Block.parameters.Motor.rPrintPosition + Block.parSw.rOffsetPrintMotor,
							Block.parameters.Motor.rMinSafePosition + Block.parSw.rOffsetPrintMotor);

	//Manage Block.Status.BlockState depending on the MachineMode
	//	PRINTERGEN_ZERO:
	//	PRINTERGEN_MANUAL:
	//	PRINTERGEN_AUTO:
	BlockStateMach;

	//Manage the General State of the BLOCK
	//	BLOCK_STOPPED:
	//	BLOCK_STOPPING:
	//	BLOCK_MANUAL:
	//	BLOCK_AUTO:
	BlockStateGen;

	//Manage the current position of the Block
	//	BLOCKP_UNDEFINED:
	//	BLOCKP_HOMING_ICLA:
	//	BLOCKP_HOMING_BAR:
	//	BLOCKP_IN_CAP:
	//	BLOCKP_IN_PRINT:
	//	BLOCKP_GOING_TO_CAP:
	//	BLOCKP_GOING_TO_PRINT:
	PreviousLogic;
	BlockStatePos;
	PosteriorLogic;

	LogOrders;
	DefineBoolPositionStatus;
	RegisterCyclesInPosState;

	BlockStatePrevious := Block.Status.BlockState;
	MachineStatePrevious :=  Block.commands.StateMode;

END_ACTION

ACTION StopMovements:

	StopBar;

END_ACTION

ACTION RegisterCyclesInPosState:

	//BlockStates to SW and times in each position
	CASE Block.Status.PositionState OF
		BLOCKP_UNDEFINED:		Block.Status.iBlockState:= 0; iTimesStateBlockUndefined := iTimesStateBlockUndefined+1;
		BLOCKP_HOMING_BAR:		Block.Status.iBlockState:= 0; iTimesStateBlockHomingBar := iTimesStateBlockHomingBar+1;
		BLOCKP_IN_CAP:			Block.Status.iBlockState:= 1; iTimesStateBlockInCap := iTimesStateBlockInCap+1;
		BLOCKP_IN_PRINT:		Block.Status.iBlockState:= 2; iTimesStateBlockPrinting := iTimesStateBlockPrinting+1;
		BLOCKP_GOING_TO_CAP:	Block.Status.iBlockState:= 4; iTimesStateBlockGoingToCap := iTimesStateBlockGoingToCap+1;
		BLOCKP_GOING_TO_PRINT:	Block.Status.iBlockState:= 5; iTimesStateBlockGoingToPrint := iTimesStateBlockGoingToPrint+1;
	END_CASE

END_ACTION

ACTION DefineBoolPositionStatus:

	Block.Status.Position.xUndefined	:= 	Block.Status.PositionState = BLOCKP_UNDEFINED;
	Block.Status.Position.xInCap    	:=	Block.Status.PositionState = BLOCKP_IN_CAP;
	Block.Status.Position.xInPrint 		:=	Block.Status.PositionState = BLOCKP_IN_PRINT;
	Block.Status.Position.xGoingToCap	:=	Block.Status.PositionState = BLOCKP_GOING_TO_CAP;
	Block.Status.Position.xGoingToPrint :=	Block.Status.PositionState = BLOCKP_GOING_TO_PRINT;

END_ACTION

ACTION ResetKnownPositions:

	xInCap:= FALSE;
	xInPrint:= FALSE;

END_ACTION

ACTION LogOrders:

	IF  Block.Status.PositionState = BLOCKP_GOING_TO_CAP AND BlockPositionPrevious <> BLOCKP_GOING_TO_CAP THEN
		LogToCapOrder;
	END_IF
	IF Block.Status.PositionState = BLOCKP_GOING_TO_PRINT AND BlockPositionPrevious <> BLOCKP_GOING_TO_PRINT THEN
		LogToPrintOrder;
	END_IF

END_ACTION
```

#### ControlState.st
```iecst
ACTION ControlState:

	// General states
	Block.Status.Motor.xBarsHoming:= AxisBK.Status.PLCopenState.Homing; //  States for Homing block
	Block.Status.Motor.rTorque := AxisBK.Status.ActTorque;
	Block.Status.Motor.ErrorID := AxisBK.Status.ErrorID;
	Block.Status.Motor.rActPosition := AxisBK.Status.ActPosition;
	Block.Status.Motor.rSpeed := AxisBK.Status.ActVelocity;
	Block.Status.Motor.rActPosition := AxisBK.Status.ActPosition;

	// Speed paramter for auto movements
	MotorDriveUnit.PulsesSpeedDevice := AxisBK.Status.ActVelocity;
	MotorDriveUnit.Calculation := CALC_SPEED_MM;
	MotorDriveUnit();
	Block.Status.Motor.rSpeed := MotorDriveUnit.SpeedDevice;

	xAnyManualMovement := AxisBK.Status.PLCopenState.ContinuousMotion AND Block.commands.Mode.xManual;
	Block.Status.xAnyManualMovement:=xAnyManualMovement;

END_ACTION
```

#### EventLog.st
```iecst
ACTION LogCriticalAlarm:

//	iReasonCritical.0 := (Block.Al.xAlrSafetySystemInBlock AND Block.Status.xEnabledMovements);
//	iReasonCritical.1 := Block.Al.xAlrDriveProtection;

	stEventLog.Source := ELOG_TYPE_SIMPLEBLOCK;
	stEventLog.Severity:= ELOG_SEVERITY_ERROR;
	stEventLog.Facility:= gIndexSimpleBlock;
	stEventLog.ErrorCode:=0;

	stEventLog.Text := 'SBlock.LogCriticalAlarm';

	IF 		iReasonCritical.0 THEN stEventLog.Text := 'SBlock. xAlrSafetySystemInBlock';
	ELSIF 	iReasonCritical.1 THEN stEventLog.Text := 'SBlock. xAlrDriveProtection';
	END_IF

	gEventLogLoader(EventData := ADR(stEventLog));

END_ACTION

ACTION LogStopAlarm:

//	// Stop Alarms. The machine goes to Automatic-Stop.
//	iReasonStop.0 := Block.Al.xAnyDriveAlarm;
//	iReasonStop.1 := Block.Al.xAlrBarMtrNoRef;
//	iReasonStop.2 := Block.Al.xAlrComBarMtr;

	stEventLog.Source := ELOG_TYPE_SIMPLEBLOCK;
	stEventLog.Severity:= ELOG_SEVERITY_ERROR;
	stEventLog.Facility:= gIndexSimpleBlock;
	stEventLog.ErrorCode:=0;

	stEventLog.Text := 'SBlock.LogStopAlarm';

	IF 		iReasonStop.0 THEN stEventLog.Text := 'SBlock. xAnyDriveAlarm';
	ELSIF 	iReasonStop.1 THEN stEventLog.Text := 'SBlock. xAlrBarMtrNoRef';
	ELSIF 	iReasonStop.2 THEN stEventLog.Text := 'SBlock. xAlrComBarMtr';
	END_IF

	gEventLogLoader(EventData := ADR(stEventLog));

END_ACTION

ACTION LogToCapOrder:

	stEventLog.Source := ELOG_TYPE_SIMPLEBLOCK;
	stEventLog.Severity:= ELOG_SEVERITY_INFO;
	stEventLog.Facility:= gIndexSimpleBlock;
	stEventLog.ErrorCode:=0;

	stEventLog.Text := 'Order to Cap BK: ';
	brsitoa(gIndexSimpleBlock, ADR(strAuxEventDesc));
	brsstrcat(ADR(stEventLog.Text), ADR(strAuxEventDesc));

	gEventLogLoader(EventData := ADR(stEventLog));

END_ACTION

ACTION LogToPrintOrder:

	stEventLog.Source := ELOG_TYPE_SIMPLEBLOCK;
	stEventLog.Severity:= ELOG_SEVERITY_INFO;
	stEventLog.Facility:= gIndexSimpleBlock;
	stEventLog.ErrorCode:=0;

	stEventLog.Text := 'Order to Print BK: ';
	brsitoa(gIndexSimpleBlock, ADR(strAuxEventDesc));
	brsstrcat(ADR(stEventLog.Text), ADR(strAuxEventDesc));

	gEventLogLoader(EventData := ADR(stEventLog));

END_ACTION

ACTION LogVertMovementOrder:

	VerMotorEventLog.Source := ELOG_TYPE_SIMPLEBLOCK;
	VerMotorEventLog.Severity:= ELOG_SEVERITY_INFO;
	VerMotorEventLog.Facility:= gIndexSimpleBlock;
	VerMotorEventLog.ErrorCode:=0;

	VerMotorEventLog.Text := 'Vert Mov Order BK: ';
	brsitoa(gIndexSimpleBlock, ADR(strAuxEventDesc));
	brsstrcat(ADR(VerMotorEventLog.Text), ADR(strAuxEventDesc));
	brsstrcat(ADR(VerMotorEventLog.Text), ADR(': '));
	brsftoa(MotorDriveUnit.PositionDesired, ADR(strAuxEventDesc));
	brsstrcat(ADR(VerMotorEventLog.Text), ADR(strAuxEventDesc));
	brsstrcat(ADR(VerMotorEventLog.Text), ADR('mm. St: '));
	brsitoa(nState, ADR(strAuxEventDesc));
	brsstrcat(ADR(VerMotorEventLog.Text), ADR(strAuxEventDesc));

	gEventLogLoader(EventData := ADR(VerMotorEventLog));

END_ACTION

ACTION LogVertInPosition:

	VerMotorEventLog.Source := ELOG_TYPE_SIMPLEBLOCK;
	VerMotorEventLog.Severity:= ELOG_SEVERITY_INFO;
	VerMotorEventLog.Facility:= gIndexSimpleBlock;
	VerMotorEventLog.ErrorCode:=0;

	VerMotorEventLog.Text := 'Vert Mov In Position BK: ';
	brsitoa(gIndexSimpleBlock, ADR(strAuxEventDesc));
	brsstrcat(ADR(VerMotorEventLog.Text), ADR(strAuxEventDesc));
	brsstrcat(ADR(VerMotorEventLog.Text), ADR(': '));
	brsftoa(MotorDriveUnit.PositionDevice, ADR(strAuxEventDesc));
	brsstrcat(ADR(VerMotorEventLog.Text), ADR(strAuxEventDesc));
	brsstrcat(ADR(VerMotorEventLog.Text), ADR('mm. St: '));
	brsitoa(nState, ADR(strAuxEventDesc));
	brsstrcat(ADR(VerMotorEventLog.Text), ADR(strAuxEventDesc));

	gEventLogLoader(EventData := ADR(VerMotorEventLog));

END_ACTION

ACTION LogHomingOrderBar:

	VerMotorEventLog.Source := ELOG_TYPE_SIMPLEBLOCK;
	VerMotorEventLog.Severity:= ELOG_SEVERITY_INFO;
	VerMotorEventLog.Facility:= gIndexSimpleBlock;
	VerMotorEventLog.ErrorCode:=0;

	VerMotorEventLog.Text := 'Homing order Vert BK: ';
	brsitoa(gIndexSimpleBlock, ADR(strAuxEventDesc));
	brsstrcat(ADR(VerMotorEventLog.Text), ADR(strAuxEventDesc));

	gEventLogLoader(EventData := ADR(VerMotorEventLog));

END_ACTION

ACTION LogHomedBar:

	VerMotorEventLog.Source := ELOG_TYPE_SIMPLEBLOCK;
	VerMotorEventLog.Severity:= ELOG_SEVERITY_INFO;
	VerMotorEventLog.Facility:= gIndexSimpleBlock;
	VerMotorEventLog.ErrorCode:=0;

	VerMotorEventLog.Text := 'Vert Motor Homed BK: ';
	brsitoa(gIndexSimpleBlock, ADR(strAuxEventDesc));
	brsstrcat(ADR(VerMotorEventLog.Text), ADR(strAuxEventDesc));

	gEventLogLoader(EventData := ADR(VerMotorEventLog));

END_ACTION
```

#### GeneralLogic.st
```iecst
ACTION PreviousLogic:

	IF NOT AxisBK.Status.HomeOK THEN
		Block.Status.Motor.xBarsHomed:= FALSE;
	END_IF

	IF Block.Status.PositionState <> BLOCKP_IN_PRINT THEN
		Block.Status.Position.xReadyToPrint := FALSE;
	END_IF

END_ACTION

ACTION PosteriorLogic:

	// Update state
	Block.Status.iBlockCaseLogicControl:=nState;

END_ACTION
```

#### LogicFunctions.st
```iecst
(* This function returns if the bar determined by the index is in the current block *)
FUNCTION AllDevicedStopped
	AllDevicedStopped := NOT AxisBK.Status.PLCopenState.ContinuousMotion AND
						NOT AxisBK.Status.PLCopenState.Stopping AND
						NOT AxisBK.Status.PLCopenState.DiscreteMotion;

END_FUNCTION
```

#### ResetAlarms.st
```iecst
ACTION ResetAlarms:

	Block.Al:= SimpleBlockAlarmsReseted;
	Block.AlSummary:= SimpleBlockAlarmsSummaryReseted;

END_ACTION
```

### Program Logical/ExtPack/SimpleBlockCtrl/SimpleBlockSim/SimpleBlockSim_v1/SimpleBlockSim (IEC)

#### BlockSim.var
```iecst
VAR
	Block : REFERENCE TO SimpleBlock;
	MotorBlock : REFERENCE TO AxisCtrl_typ;
	SimBlock : REFERENCE TO SimBlock_typ;
	fbWriteRefSignal : MC_BR_WriteParID;
	iRefSignalState : USINT;
	AxisRef : UDINT;
	StatusNcAccess : UINT;
	uiValueRef : DINT;
	TimesExcecHoming : USINT;
END_VAR
```

### Program Logical/ExtPack/SimpleBlockCtrl/SimpleBlockSim/SimpleBlockSim_v1/InitSimpleBlockSim (IEC)

#### Main.st - Init, cyclic, exit code
```iecst
PROGRAM _CYCLIC

	iSimpleBlockSimIndex:= 1;

END_PROGRAM
```

### SimpleBlockSim.var
```iecst
VAR
	iSimpleBlockSimIndex : USINT;
END_VAR
```

### BlockSim.typ
```iecst
TYPE
	SimSimpleBlockCommands_typ : 	STRUCT
		DelayHomingBar : BOOL; (*With this activated, the SimBlock waits to home the bars until this signal is released*)
	END_STRUCT;
	SimSimpleBlockParameters_typ : 	STRUCT
		New_Member : BOOL;
	END_STRUCT;
	SimSimpleBlock_typ : 	STRUCT
		Commands : SimSimpleBlockCommands_typ;
		Parameters : SimSimpleBlockParameters_typ;
	END_STRUCT;
END_TYPE
```
